KUKA KRL program: MyProgram_124().src

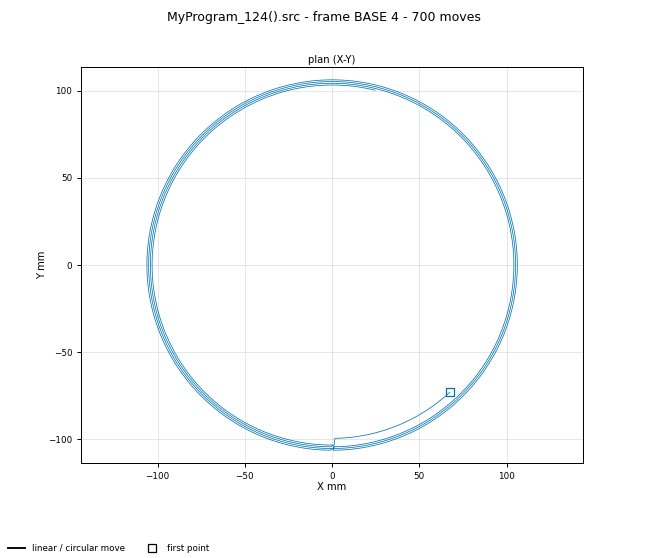
[picture p0: tool path of MyProgram_124().src in frame BASE 4, 700 of 700 moves have a stored position in this frame; points joined in program order, loops and branches not executed]
&ACCESS RVP
&REL 1
&PARAM TEMPLATE = C:\KRC\Roboter\Template\vorgabe
&PARAM EDITMASK = *
DEF MyProgram_124()
; ---- Setting reference (Base) ----
$BASE = BASE_DATA[4]

; --------------------------
; ---- Setting tool (TCP) ----
$TOOL = TOOL_DATA[3]
; --------------------------

$VEL.CP = VEL_APROX_PRINT
Startdeposition()
$VEL.CP = VEL_PRINT
LIN {X 67.4636,Y -72.9151,Z 103,A -51.9961,B 24.9391,C -1.8028,E1 25.1077,E2 497.4549} C_DIS
LIN {X 64.8778,Y -75.2264,Z 103,A -54.0592,B 24.9396,C -1.7957,E1 25.1034,E2 499.5265} C_DIS
LIN {X 62.0723,Y -77.5576,Z 103,A -56.1658,B 24.9399,C -1.791,E1 25.0988,E2 501.6364} C_DIS
LIN {X 59.4843,Y -79.5578,Z 103,A -57.817,B 24.9395,C -1.7961,E1 25.0952,E2 503.2694} C_DIS
LIN {X 57.5377,Y -80.9767,Z 103,A -59.2001,B 24.9397,C -1.7935,E1 25.092,E2 504.6539} C_DIS
LIN {X 55.1858,Y -82.5995,Z 103,A -61.0068,B 24.9403,C -1.784,E1 25.0878,E2 506.4769} C_DIS
LIN {X 52.4682,Y -84.3499,Z 103,A -62.7627,B 24.9403,C -1.7846,E1 25.0837,E2 508.2256} C_DIS
LIN {X 50.0146,Y -85.8293,Z 103,A -64.3819,B 24.9404,C -1.7828,E1 25.0798,E2 509.8441} C_DIS
LIN {X 47.8461,Y -87.0565,Z 103,A -65.9289,B 24.9409,C -1.7761,E1 25.076,E2 511.4025} C_DIS
LIN {X 45.0141,Y -88.5525,Z 103,A -67.6742,B 24.9409,C -1.7769,E1 25.0717,E2 513.141} C_DIS
LIN {X 42.0972,Y -89.9758,Z 103,A -69.5826,B 24.9411,C -1.7725,E1 25.0669,E2 515.0548} C_DIS
LIN {X 39.1268,Y -91.3084,Z 103,A -71.5179,B 24.9415,C -1.7674,E1 25.0619,E2 516.9974} C_DIS
LIN {X 36.1356,Y -92.5313,Z 103,A -73.2136,B 24.9412,C -1.7713,E1 25.0575,E2 518.6802} C_DIS
LIN {X 33.7277,Y -93.4362,Z 103,A -74.6858,B 24.9413,C -1.7697,E1 25.0537,E2 520.153} C_DIS
LIN {X 31.1034,Y -94.3433,Z 103,A -76.4427,B 24.9418,C -1.7618,E1 25.049,E2 521.9253} C_DIS
LIN {X 28.0406,Y -95.2971,Z 103,A -78.1345,B 24.9416,C -1.7657,E1 25.0445,E2 523.6049} C_DIS
LIN {X 25.3105,Y -96.06,Z 103,A -79.7633,B 24.9416,C -1.7641,E1 25.0401,E2 525.2347} C_DIS
LIN {X 22.5573,Y -96.7418,Z 103,A -81.5,B 24.942,C -1.7587,E1 25.0354,E2 526.9817} C_DIS
LIN {X 19.9429,Y -97.3142,Z 103,A -83.0396,B 24.9421,C -1.7575,E1 25.0312,E2 528.5221} C_DIS
LIN {X 16.9823,Y -97.8762,Z 103,A -84.8399,B 24.9424,C -1.7538,E1 25.0262,E2 530.3294} C_DIS
LIN {X 13.8632,Y -98.3646,Z 103,A -86.5531,B 24.9422,C -1.7565,E1 25.0215,E2 532.0345} C_DIS
LIN {X 10.9392,Y -98.7343,Z 103,A -88.1902,B 24.9421,C -1.7578,E1 25.017,E2 533.6673} C_DIS
LIN {X 8.1007,Y -99.006,Z 103,A -89.9343,B 24.9424,C -1.7533,E1 25.0121,E2 535.4211} C_DIS
LIN {X 4.8754,Y -99.2188,Z 103,A -91.8612,B 24.9426,C -1.7502,E1 25.0067,E2 537.3547} C_DIS
LIN {X 1.6447,Y -99.3232,Z 103,A -93.5925,B 24.9423,C -1.7545,E1 25.0019,E2 539.0753} C_DIS
LIN {X 1.6447,Y -99.3232,Z 103,A -93.5925,B 24.9423,C -1.7545,E1 25.0019,E2 539.0753} C_DIS
Enddeposition()
LIN {X 0.7394,Y -106.1621,Z 104,A -93.403,B 24.9477,C -1.6702,E1 25.0019,E2 539.0857} C_DIS
Startdeposition()
$VEL.CP = VEL_PRINT
LIN {X 4.4145,Y -106.0742,Z 104,A -91.2125,B 24.9472,C -1.6792,E1 25.008,E2 536.8744} C_DIS
LIN {X 7.8102,Y -105.8803,Z 104,A -89.2631,B 24.9468,C -1.6846,E1 25.0135,E2 534.913} C_DIS
LIN {X 10.7746,Y -105.6181,Z 104,A -87.8003,B 24.9471,C -1.6797,E1 25.0175,E2 533.4628} C_DIS
LIN {X 14.6548,Y -105.15,Z 104,A -85.7013,B 24.9471,C -1.6806,E1 25.0233,E2 531.3633} C_DIS
LIN {X 18.1507,Y -104.6049,Z 104,A -83.6459,B 24.9466,C -1.688,E1 25.0291,E2 529.2925} C_DIS
LIN {X 20.7123,Y -104.128,Z 104,A -82.2422,B 24.9466,C -1.6891,E1 25.0329,E2 527.8878} C_DIS
LIN {X 23.5206,Y -103.5284,Z 104,A -80.7997,B 24.9467,C -1.6861,E1 25.0368,E2 526.4542} C_DIS
LIN {X 25.7967,Y -102.9862,Z 104,A -79.5774,B 24.9467,C -1.6857,E1 25.0401,E2 525.2348} C_DIS
LIN {X 28.3163,Y -102.3221,Z 104,A -78.0325,B 24.9463,C -1.6929,E1 25.0443,E2 523.6752} C_DIS
LIN {X 30.8189,Y -101.5964,Z 104,A -76.7716,B 24.9466,C -1.6885,E1 25.0477,E2 522.427} C_DIS
LIN {X 33.6539,Y -100.6911,Z 104,A -75.0798,B 24.9462,C -1.6941,E1 25.0522,E2 520.7253} C_DIS
LIN {X 36.9909,Y -99.5153,Z 104,A -73.1238,B 24.9459,C -1.6985,E1 25.0573,E2 518.7628} C_DIS
LIN {X 40.6287,Y -98.0864,Z 104,A -71.1625,B 24.9461,C -1.6953,E1 25.0624,E2 516.8135} C_DIS
LIN {X 43.0236,Y -97.0598,Z 104,A -69.761,B 24.9461,C -1.6972,E1 25.066,E2 515.4108} C_DIS
LIN {X 45.3926,Y -95.9747,Z 104,A -68.3595,B 24.9459,C -1.6993,E1 25.0695,E2 514.0081} C_DIS
LIN {X 48.0641,Y -94.6632,Z 104,A -66.7592,B 24.9457,C -1.7017,E1 25.0735,E2 512.4063} C_DIS
LIN {X 51.1925,Y -93.0106,Z 104,A -64.7153,B 24.9452,C -1.7106,E1 25.0786,E2 510.3472} C_DIS
LIN {X 53.7785,Y -91.5378,Z 104,A -63.2568,B 24.9454,C -1.7074,E1 25.0821,E2 508.9008} C_DIS
LIN {X 56.0305,Y -90.1768,Z 104,A -61.8515,B 24.9452,C -1.7094,E1 25.0854,E2 507.4951} C_DIS
LIN {X 59.2904,Y -88.0678,Z 104,A -59.7558,B 24.945,C -1.7136,E1 25.0903,E2 505.3965} C_DIS
LIN {X 61.4338,Y -86.5862,Z 104,A -58.356,B 24.9448,C -1.7162,E1 25.0935,E2 503.9954} C_DIS
LIN {X 63.5403,Y -85.0524,Z 104,A -56.9295,B 24.9446,C -1.72,E1 25.0967,E2 502.565} C_DIS
LIN {X 65.6084,Y -83.4675,Z 104,A -55.5565,B 24.9445,C -1.7216,E1 25.0998,E2 501.1931} C_DIS
LIN {X 67.6371,Y -81.8322,Z 104,A -54.1568,B 24.9443,C -1.7245,E1 25.1028,E2 499.792} C_DIS
LIN {X 69.625,Y -80.1477,Z 104,A -52.7579,B 24.9441,C -1.7274,E1 25.1058,E2 498.3917} C_DIS
LIN {X 71.5709,Y -78.4149,Z 104,A -51.3584,B 24.9439,C -1.7304,E1 25.1087,E2 496.9908} C_DIS
LIN {X 74.4086,Y -75.7274,Z 104,A -49.4414,B 24.9441,C -1.7272,E1 25.1125,E2 495.0891} C_DIS
LIN {X 76.2447,Y -73.8785,Z 104,A -48.0425,B 24.9439,C -1.7304,E1 25.1153,E2 493.6888} C_DIS
LIN {X 77.7844,Y -72.258,Z 104,A -46.6614,B 24.9432,C -1.7409,E1 25.1179,E2 492.2889} C_DIS
LIN {X 79.5343,Y -70.3273,Z 104,A -45.2623,B 24.943,C -1.7441,E1 25.1205,E2 490.8884} C_DIS
LIN {X 81.5346,Y -67.9952,Z 104,A -43.8429,B 24.9434,C -1.7383,E1 25.1231,E2 489.4892} C_DIS
LIN {X 82.8893,Y -66.34,Z 104,A -42.4537,B 24.9425,C -1.7514,E1 25.1256,E2 488.0756} C_DIS
LIN {X 84.4924,Y -64.2859,Z 104,A -41.068,B 24.9423,C -1.7543,E1 25.1279,E2 486.6896} C_DIS
LIN {X 86.0446,Y -62.193,Z 104,A -39.6701,B 24.9421,C -1.7578,E1 25.1302,E2 485.2901} C_DIS
LIN {X 87.79,Y -59.7006,Z 104,A -38.061,B 24.9419,C -1.761,E1 25.1328,E2 483.6814} C_DIS
LIN {X 89.8926,Y -56.4855,Z 104,A -36.1587,B 24.9419,C -1.7595,E1 25.1356,E2 481.7921} C_DIS
LIN {X 91.0633,Y -54.5812,Z 104,A -34.7784,B 24.9413,C -1.7705,E1 25.1377,E2 480.3931} C_DIS
LIN {X 92.5559,Y -52.0066,Z 104,A -33.1821,B 24.941,C -1.7747,E1 25.1399,E2 478.7949} C_DIS
LIN {X 94.2389,Y -48.8944,Z 104,A -31.1438,B 24.9402,C -1.786,E1 25.1426,E2 476.7409} C_DIS
LIN {X 95.5708,Y -46.2332,Z 104,A -29.6891,B 24.9403,C -1.7842,E1 25.1444,E2 475.298} C_DIS
LIN {X 96.6964,Y -43.83,Z 104,A -28.283,B 24.9401,C -1.7875,E1 25.146,E2 473.8919} C_DIS
LIN {X 97.7242,Y -41.488,Z 104,A -26.8064,B 24.9396,C -1.7959,E1 25.1476,E2 472.4035} C_DIS
LIN {X 98.9185,Y -38.554,Z 104,A -25.1568,B 24.9394,C -1.7985,E1 25.1493,E2 470.7568} C_DIS
LIN {X 99.9618,Y -35.7669,Z 104,A -23.6014,B 24.9392,C -1.8013,E1 25.1508,E2 469.2036} C_DIS
LIN {X 100.9235,Y -32.9506,Z 104,A -22.0063,B 24.9389,C -1.8059,E1 25.1522,E2 467.6066} C_DIS
LIN {X 102.0679,Y -29.2135,Z 104,A -19.9111,B 24.9385,C -1.812,E1 25.1539,E2 465.5091} C_DIS
LIN {X 102.9862,Y -25.7967,Z 104,A -17.8737,B 24.9377,C -1.8236,E1 25.1554,E2 463.4561} C_DIS
LIN {X 103.5883,Y -23.2615,Z 104,A -16.4771,B 24.9374,C -1.8277,E1 25.1562,E2 462.0579} C_DIS
LIN {X 104.1964,Y -20.3566,Z 104,A -15.0246,B 24.9374,C -1.8263,E1 25.157,E2 460.617} C_DIS
LIN {X 104.666,Y -17.7854,Z 104,A -13.6266,B 24.9372,C -1.8303,E1 25.1577,E2 459.2178} C_DIS
LIN {X 105.2497,Y -13.9209,Z 104,A -11.7135,B 24.9373,C -1.8287,E1 25.1585,E2 457.3199} C_DIS
LIN {X 105.5491,Y -11.4338,Z 104,A -10.118,B 24.9363,C -1.8436,E1 25.159,E2 455.6986} C_DIS
LIN {X 105.8803,Y -7.8102,Z 104,A -8.0982,B 24.9357,C -1.8524,E1 25.1595,E2 453.6701} C_DIS
LIN {X 106.0401,Y -5.2094,Z 104,A -6.7017,B 24.9354,C -1.8565,E1 25.1597,E2 452.2721} C_DIS
LIN {X 106.1531,Y -1.6731,Z 104,A -4.7932,B 24.935,C -1.8627,E1 25.1597,E2 450.3604} C_DIS
LIN {X 106.136,Y 2.6055,Z 104,A -2.5124,B 24.9345,C -1.8689,E1 25.1597,E2 448.0787} C_DIS
LIN {X 106.0401,Y 5.2094,Z 104,A -1.1158,B 24.9342,C -1.873,E1 25.1595,E2 446.6806} C_DIS
LIN {X 105.8803,Y 7.8102,Z 104,A 0.2806,B 24.934,C -1.8771,E1 25.1592,E2 445.2829} C_DIS
LIN {X 105.5211,Y 11.7021,Z 104,A 2.4327,B 24.9333,C -1.8857,E1 25.1586,E2 443.1232} C_DIS
LIN {X 105.0188,Y 15.5781,Z 104,A 4.3294,B 24.9335,C -1.8831,E1 25.1579,E2 441.2437} C_DIS
LIN {X 104.6049,Y 18.1507,Z 104,A 5.8673,B 24.9328,C -1.8933,E1 25.1572,E2 439.6909} C_DIS
LIN {X 104.0535,Y 21.0751,Z 104,A 7.3213,B 24.9329,C -1.8917,E1 25.1564,E2 438.249} C_DIS
LIN {X 103.2072,Y 24.8908,Z 104,A 9.2641,B 24.9329,C -1.8911,E1 25.1552,E2 436.3189} C_DIS
LIN {X 102.6619,Y 27.0586,Z 104,A 10.7562,B 24.9318,C -1.9071,E1 25.1542,E2 434.7977} C_DIS
LIN {X 101.8958,Y 29.8097,Z 104,A 12.0237,B 24.9323,C -1.9,E1 25.1532,E2 433.5542} C_DIS
LIN {X 101.2105,Y 32.0633,Z 104,A 13.4091,B 24.9317,C -1.9088,E1 25.152,E2 432.156} C_DIS
LIN {X 100.3932,Y 34.5375,Z 104,A 14.9476,B 24.931,C -1.9187,E1 25.1506,E2 430.6028} C_DIS
LIN {X 99.3842,Y 37.3372,Z 104,A 16.4024,B 24.9311,C -1.917,E1 25.1493,E2 429.1602} C_DIS
LIN {X 98.5433,Y 39.5062,Z 104,A 17.6053,B 24.9311,C -1.9184,E1 25.148,E2 427.9607} C_DIS
LIN {X 97.5296,Y 41.9459,Z 104,A 19.0045,B 24.9308,C -1.9214,E1 25.1465,E2 426.562} C_DIS
LIN {X 96.5245,Y 44.2115,Z 104,A 20.5441,B 24.9299,C -1.9338,E1 25.1447,E2 425.0014} C_DIS
LIN {X 95.4104,Y 46.567,Z 104,A 21.7939,B 24.9301,C -1.9311,E1 25.1432,E2 423.7647} C_DIS
LIN {X 94.2389,Y 48.8944,Z 104,A 23.1917,B 24.9298,C -1.9347,E1 25.1414,E2 422.366} C_DIS
LIN {X 92.83,Y 51.5158,Z 104,A 24.7883,B 24.9295,C -1.9387,E1 25.1393,E2 420.7683} C_DIS
LIN {X 90.8019,Y 55.0114,Z 104,A 26.9328,B 24.9292,C -1.943,E1 25.1363,E2 418.6247} C_DIS
LIN {X 88.9926,Y 57.896,Z 104,A 28.7841,B 24.9288,C -1.9483,E1 25.1335,E2 416.7701} C_DIS
LIN {X 87.3336,Y 60.3667,Z 104,A 30.3816,B 24.9286,C -1.9521,E1 25.131,E2 415.1715} C_DIS
LIN {X 85.2749,Y 63.2442,Z 104,A 32.2808,B 24.9282,C -1.9564,E1 25.1278,E2 413.2714} C_DIS
LIN {X 83.6971,Y 65.3179,Z 104,A 33.6798,B 24.928,C -1.9595,E1 25.1255,E2 411.8716} C_DIS
LIN {X 81.8322,Y 67.6371,Z 104,A 35.2776,B 24.9278,C -1.963,E1 25.1226,E2 410.273} C_DIS
LIN {X 80.2103,Y 69.5532,Z 104,A 36.6598,B 24.9274,C -1.9673,E1 25.1201,E2 408.8869} C_DIS
LIN {X 78.6653,Y 71.298,Z 104,A 37.8771,B 24.9274,C -1.9684,E1 25.1179,E2 407.6724} C_DIS
LIN {X 76.8918,Y 73.2071,Z 104,A 39.2766,B 24.9271,C -1.9713,E1 25.1152,E2 406.2723} C_DIS
LIN {X 74.8086,Y 75.3323,Z 104,A 40.6937,B 24.9275,C -1.9668,E1 25.1124,E2 404.8717} C_DIS
LIN {X 73.2071,Y 76.8918,Z 104,A 42.0765,B 24.9267,C -1.9767,E1 25.1096,E2 403.4713} C_DIS
LIN {X 71.0221,Y 78.9123,Z 104,A 43.6753,B 24.9265,C -1.9797,E1 25.1063,E2 401.8719} C_DIS
LIN {X 68.0694,Y 81.4729,Z 104,A 45.8349,B 24.9261,C -1.9859,E1 25.1017,E2 399.706} C_DIS
LIN {X 65.3179,Y 83.6971,Z 104,A 47.8193,B 24.9256,C -1.9925,E1 25.0974,E2 397.7134} C_DIS
LIN {X 63.2442,Y 85.2749,Z 104,A 49.0899,B 24.9258,C -1.9894,E1 25.0945,E2 396.4548} C_DIS
LIN {X 61.1324,Y 86.8013,Z 104,A 50.4796,B 24.9257,C -1.9911,E1 25.0914,E2 395.0658} C_DIS
LIN {X 58.6746,Y 88.4793,Z 104,A 52.08,B 24.9255,C -1.9935,E1 25.0877,E2 393.4651} C_DIS
LIN {X 56.4855,Y 89.8926,Z 104,A 53.5325,B 24.9252,C -1.9976,E1 25.0842,E2 392.0076} C_DIS
LIN {X 53.4596,Y 91.7262,Z 104,A 55.5266,B 24.9247,C -2.0039,E1 25.0794,E2 390.0048} C_DIS
LIN {X 50.0472,Y 93.6318,Z 104,A 57.6296,B 24.9245,C -2.0066,E1 25.0743,E2 387.9015} C_DIS
LIN {X 47.7343,Y 94.8318,Z 104,A 58.8901,B 24.9248,C -2.0024,E1 25.0712,E2 386.6544} C_DIS
LIN {X 45.3926,Y 95.9747,Z 104,A 60.4347,B 24.9243,C -2.0098,E1 25.0673,E2 385.0964} C_DIS
LIN {X 42.6841,Y 97.2078,Z 104,A 61.8947,B 24.9246,C -2.0057,E1 25.0636,E2 383.6497} C_DIS
LIN {X 39.9794,Y 98.3507,Z 104,A 63.5207,B 24.9243,C -2.009,E1 25.0594,E2 382.0195} C_DIS
LIN {X 36.9909,Y 99.5153,Z 104,A 65.3455,B 24.9239,C -2.0145,E1 25.0546,E2 380.1857} C_DIS
LIN {X 34.1866,Y 100.5115,Z 104,A 66.8064,B 24.9242,C -2.01,E1 25.0508,E2 378.7384} C_DIS
LIN {X 31.6232,Y 101.347,Z 104,A 68.32,B 24.924,C -2.0135,E1 25.0467,E2 377.2192} C_DIS
LIN {X 28.6727,Y 102.2212,Z 104,A 70.0997,B 24.9235,C -2.0195,E1 25.0419,E2 375.4283} C_DIS
LIN {X 25.7967,Y 102.9862,Z 104,A 71.6633,B 24.9235,C -2.0187,E1 25.0377,E2 373.8689} C_DIS
LIN {X 23.2615,Y 103.5883,Z 104,A 72.9259,B 24.924,C -2.0137,E1 25.0343,E2 372.62} C_DIS
LIN {X 20.7123,Y 104.128,Z 104,A 74.473,B 24.9235,C -2.02,E1 25.03,E2 371.06} C_DIS
LIN {X 17.7854,Y 104.666,Z 104,A 75.9356,B 24.9239,C -2.0149,E1 25.026,E2 369.611} C_DIS
LIN {X 15.0661,Y 105.0916,Z 104,A 77.3709,B 24.9239,C -2.0133,E1 25.0221,E2 368.1808} C_DIS
LIN {X 12.6898,Y 105.4054,Z 104,A 78.561,B 24.9243,C -2.0094,E1 25.0188,E2 367.0007} C_DIS
LIN {X 10.4063,Y 105.6567,Z 104,A 80.0948,B 24.9234,C -2.0213,E1 25.0145,E2 365.44} C_DIS
LIN {X 7.8102,Y 105.8803,Z 104,A 81.5009,B 24.9234,C -2.0213,E1 25.0106,E2 364.0343} C_DIS
LIN {X 5.2094,Y 106.0401,Z 104,A 82.9074,B 24.9234,C -2.0213,E1 25.0066,E2 362.6285} C_DIS
LIN {X 1.8879,Y 106.1492,Z 104,A 84.6484,B 24.9236,C -2.0191,E1 25.0018,E2 360.8931} C_DIS
LIN {X -1.6731,Y 106.1531,Z 104,A 86.4353,B 24.924,C -2.0133,E1 24.9968,E2 359.1198} C_DIS
LIN {X -4.2778,Y 106.0801,Z 104,A 87.7061,B 24.9244,C -2.0076,E1 24.9933,E2 357.8624} C_DIS
LIN {X -6.8798,Y 105.9432,Z 104,A 89.2303,B 24.9241,C -2.0117,E1 24.9891,E2 356.328} C_DIS
LIN {X -9.4777,Y 105.7424,Z 104,A 90.704,B 24.924,C -2.0137,E1 24.9849,E2 354.8489} C_DIS
LIN {X -12.9961,Y 105.3695,Z 104,A 92.7585,B 24.9236,C -2.0182,E1 24.9792,E2 352.7824} C_DIS
LIN {X -15.5781,Y 105.0188,Z 104,A 94.0241,B 24.9241,C -2.0118,E1 24.9758,E2 351.5309} C_DIS
LIN {X -18.5419,Y 104.5345,Z 104,A 95.6379,B 24.9242,C -2.0104,E1 24.9713,E2 349.9189} C_DIS
LIN {X -22.3504,Y 103.787,Z 104,A 97.563,B 24.9248,C -2.0021,E1 24.9661,E2 348.0113} C_DIS
LIN {X -24.531,Y 103.295,Z 104,A 98.9549,B 24.9244,C -2.0081,E1 24.9623,E2 346.6032} C_DIS
LIN {X -27.0586,Y 102.6619,Z 104,A 100.364,B 24.9244,C -2.0068,E1 24.9585,E2 345.1952} C_DIS
LIN {X -29.9249,Y 101.8616,Z 104,A 101.7911,B 24.9251,C -1.9983,E1 24.9547,E2 343.7862} C_DIS
LIN {X -32.0633,Y 101.2105,Z 104,A 103.3676,B 24.9242,C -2.0111,E1 24.9504,E2 342.1765} C_DIS
LIN {X -34.887,Y 100.2706,Z 104,A 104.7938,B 24.9248,C -2.0022,E1 24.9467,E2 340.7686} C_DIS
LIN {X -38.554,Y 98.9185,Z 104,A 106.726,B 24.9255,C -1.9927,E1 24.9417,E2 338.8551} C_DIS
LIN {X -40.7938,Y 98.0168,Z 104,A 108.2418,B 24.9251,C -1.9989,E1 24.9377,E2 337.321} C_DIS
LIN {X -43.0236,Y 97.0598,Z 104,A 109.6727,B 24.9249,C -2.0016,E1 24.934,E2 335.8803} C_DIS
LIN {X -45.3926,Y 95.9747,Z 104,A 110.9409,B 24.9254,C -1.9942,E1 24.9308,E2 334.6266} C_DIS
LIN {X -48.0641,Y 94.6632,Z 104,A 112.5526,B 24.9256,C -1.9918,E1 24.9268,E2 333.0162} C_DIS
LIN {X -51.1925,Y 93.0106,Z 104,A 114.6121,B 24.9254,C -1.9942,E1 24.9217,E2 330.9453} C_DIS
LIN {X -54.5812,Y 91.0633,Z 104,A 116.5866,B 24.9261,C -1.9854,E1 24.917,E2 328.9859} C_DIS
LIN {X -57.1113,Y 89.4963,Z 104,A 118.0161,B 24.9268,C -1.9757,E1 24.9137,E2 327.5748} C_DIS
LIN {X -59.2904,Y 88.0678,Z 104,A 119.612,B 24.9265,C -1.9801,E1 24.9099,E2 325.9632} C_DIS
LIN {X -61.4338,Y 86.5862,Z 104,A 121.0241,B 24.9267,C -1.9775,E1 24.9067,E2 324.5525} C_DIS
LIN {X -64.5792,Y 84.2663,Z 104,A 123.1434,B 24.927,C -1.9735,E1 24.9019,E2 322.4353} C_DIS
LIN {X -67.3522,Y 82.0689,Z 104,A 125.2047,B 24.9269,C -1.9749,E1 24.8974,E2 320.3627} C_DIS
LIN {X -69.346,Y 80.3913,Z 104,A 126.6177,B 24.9271,C -1.972,E1 24.8944,E2 318.9512} C_DIS
LIN {X -71.5709,Y 78.4149,Z 104,A 128.0891,B 24.9277,C -1.9633,E1 24.8914,E2 317.4946} C_DIS
LIN {X -74.1452,Y 75.9877,Z 104,A 130.1963,B 24.9275,C -1.9661,E1 24.8871,E2 315.372} C_DIS
LIN {X -76.2447,Y 73.8785,Z 104,A 131.6232,B 24.9283,C -1.9556,E1 24.8844,E2 313.9641} C_DIS
LIN {X -78.6653,Y 71.298,Z 104,A 133.6864,B 24.9283,C -1.9565,E1 24.8805,E2 311.8898} C_DIS
LIN {X -80.3913,Y 69.346,Z 104,A 134.9937,B 24.9288,C -1.9492,E1 24.8781,E2 310.5939} C_DIS
LIN {X -82.0689,Y 67.3522,Z 104,A 136.3717,B 24.9291,C -1.9445,E1 24.8756,E2 309.2208} C_DIS
LIN {X -83.9232,Y 65.0245,Z 104,A 137.803,B 24.9299,C -1.9338,E1 24.8732,E2 307.8081} C_DIS
LIN {X -85.2749,Y 63.2442,Z 104,A 139.2004,B 24.9296,C -1.9375,E1 24.8708,E2 306.3951} C_DIS
LIN {X -86.8013,Y 61.1324,Z 104,A 140.7581,B 24.9295,C -1.9392,E1 24.8683,E2 304.8257} C_DIS
LIN {X -88.9926,Y 57.896,Z 104,A 142.8804,B 24.9299,C -1.9338,E1 24.865,E2 302.7058} C_DIS
LIN {X -90.579,Y 55.3781,Z 104,A 144.3533,B 24.9306,C -1.9244,E1 24.8629,E2 301.2478} C_DIS
LIN {X -92.3753,Y 52.33,Z 104,A 146.2751,B 24.9309,C -1.9193,E1 24.8602,E2 299.3282} C_DIS
LIN {X -93.8043,Y 49.7195,Z 104,A 147.7073,B 24.9317,C -1.9083,E1 24.8583,E2 297.9147} C_DIS
LIN {X -94.8318,Y 47.7343,Z 104,A 149.1055,B 24.9315,C -1.9117,E1 24.8565,E2 296.5009} C_DIS
LIN {X -96.131,Y 45.0569,Z 104,A 150.5383,B 24.9323,C -1.9006,E1 24.8548,E2 295.0868} C_DIS
LIN {X -97.0598,Y 43.0236,Z 104,A 152.1061,B 24.9316,C -1.91,E1 24.853,E2 293.4878} C_DIS
LIN {X -98.5776,Y 39.422,Z 104,A 154.06,B 24.9325,C -1.8979,E1 24.8509,E2 291.5519} C_DIS
LIN {X -99.5154,Y 36.9909,Z 104,A 155.6192,B 24.9324,C -1.8992,E1 24.8494,E2 289.981} C_DIS
LIN {X -100.8094,Y 33.3029,Z 104,A 157.5996,B 24.9332,C -1.8879,E1 24.8476,E2 288.0163} C_DIS
LIN {X -101.7485,Y 30.306,Z 104,A 159.2508,B 24.9337,C -1.881,E1 24.8462,E2 286.3719} C_DIS
LIN {X -102.4187,Y 27.9588,Z 104,A 160.6325,B 24.9338,C -1.8792,E1 24.8452,E2 284.9866} C_DIS
LIN {X -103.3784,Y 24.1701,Z 104,A 162.5727,B 24.9347,C -1.8663,E1 24.8439,E2 283.0658} C_DIS
LIN {X -103.8659,Y 21.9886,Z 104,A 164.0947,B 24.9342,C -1.8739,E1 24.843,E2 281.5167} C_DIS
LIN {X -104.4398,Y 19.0685,Z 104,A 165.5887,B 24.9348,C -1.8647,E1 24.8422,E2 280.0357} C_DIS
LIN {X -105.0188,Y 15.5781,Z 104,A 167.5117,B 24.9352,C -1.859,E1 24.8414,E2 278.1149} C_DIS
LIN {X -105.4126,Y 12.6282,Z 104,A 168.9452,B 24.936,C -1.8476,E1 24.8409,E2 276.7001} C_DIS
LIN {X -105.6567,Y 10.4063,Z 104,A 170.4872,B 24.9354,C -1.8558,E1 24.8404,E2 275.1291} C_DIS
LIN {X -105.8803,Y 7.8102,Z 104,A 171.9034,B 24.9357,C -1.8517,E1 24.8401,E2 273.7143} C_DIS
LIN {X -106.0401,Y 5.2094,Z 104,A 173.3197,B 24.936,C -1.8475,E1 24.8399,E2 272.2995} C_DIS
LIN {X -106.136,Y 2.6055,Z 104,A 174.5924,B 24.9367,C -1.8381,E1 24.8399,E2 271.0416} C_DIS
LIN {X -106.1663,Y -0.3058,Z 104,A 176.2085,B 24.9369,C -1.8346,E1 24.8398,E2 269.4239} C_DIS
LIN {X -106.0801,Y -4.2778,Z 104,A 178.1502,B 24.9379,C -1.8204,E1 24.8399,E2 267.5045} C_DIS
LIN {X -105.9432,Y -6.8798,Z 104,A 179.5665,B 24.9382,C -1.8162,E1 24.8402,E2 266.0896} C_DIS
LIN {X -105.7424,Y -9.4777,Z 104,A -178.8337,B 24.938,C -1.8188,E1 24.8405,E2 264.4741} C_DIS
LIN {X -105.478,Y -12.0699,Z 104,A -177.361,B 24.9381,C -1.8167,E1 24.841,E2 262.9975} C_DIS
LIN {X -105.0188,Y -15.5781,Z 104,A -175.4949,B 24.9387,C -1.8091,E1 24.8417,E2 261.1386} C_DIS
LIN {X -104.6049,Y -18.1507,Z 104,A -173.9358,B 24.9386,C -1.8102,E1 24.8424,E2 259.5674} C_DIS
LIN {X -104.128,Y -20.7123,Z 104,A -172.5134,B 24.9388,C -1.8064,E1 24.8432,E2 258.1458} C_DIS
LIN {X -103.5883,Y -23.2615,Z 104,A -171.1041,B 24.9391,C -1.8022,E1 24.844,E2 256.7383} C_DIS
LIN {X -102.9862,Y -25.7967,Z 104,A -169.8317,B 24.9397,C -1.7929,E1 24.8449,E2 255.4804} C_DIS
LIN {X -102.3221,Y -28.3163,Z 104,A -168.2727,B 24.9397,C -1.7942,E1 24.846,E2 253.9093} C_DIS
LIN {X -101.5964,Y -30.8189,Z 104,A -167.0005,B 24.9403,C -1.785,E1 24.847,E2 252.6517} C_DIS
LIN {X -100.6911,Y -33.6539,Z 104,A -165.3839,B 24.9406,C -1.7806,E1 24.8484,E2 251.0363} C_DIS
LIN {X -99.5153,Y -36.9909,Z 104,A -163.3114,B 24.9406,C -1.781,E1 24.8504,E2 248.9513} C_DIS
LIN {X -98.0864,Y -40.6287,Z 104,A -161.339,B 24.9413,C -1.7698,E1 24.8524,E2 246.9946} C_DIS
LIN {X -97.0598,Y -43.0236,Z 104,A -159.9039,B 24.9415,C -1.7668,E1 24.854,E2 245.5587} C_DIS
LIN {X -95.9747,Y -45.3926,Z 104,A -158.5092,B 24.9418,C -1.7624,E1 24.8557,E2 244.1669} C_DIS
LIN {X -94.6632,Y -48.0641,Z 104,A -156.8933,B 24.9421,C -1.7583,E1 24.8577,E2 242.5521} C_DIS
LIN {X -93.0106,Y -51.1925,Z 104,A -154.8294,B 24.9421,C -1.7588,E1 24.8604,E2 240.4761} C_DIS
LIN {X -91.5378,Y -53.7785,Z 104,A -153.3321,B 24.9426,C -1.7504,E1 24.8625,E2 238.9908} C_DIS
LIN {X -89.4963,Y -57.1113,Z 104,A -151.419,B 24.9434,C -1.7376,E1 24.8653,E2 237.0986} C_DIS
LIN {X -88.0678,Y -59.2904,Z 104,A -149.8211,B 24.9432,C -1.7411,E1 24.8678,E2 235.4843} C_DIS
LIN {X -86.5862,Y -61.4338,Z 104,A -148.4075,B 24.9434,C -1.7379,E1 24.8701,E2 234.0714} C_DIS
LIN {X -84.8783,Y -63.7721,Z 104,A -146.9035,B 24.9438,C -1.7318,E1 24.8725,E2 232.5746} C_DIS
LIN {X -83.4675,Y -65.6084,Z 104,A -145.58,B 24.9438,C -1.7316,E1 24.8748,E2 231.2455} C_DIS
LIN {X -81.8322,Y -67.6371,Z 104,A -144.1664,B 24.944,C -1.7285,E1 24.8773,E2 229.8325} C_DIS
LIN {X -80.1477,Y -69.625,Z 104,A -142.7535,B 24.9442,C -1.7255,E1 24.8799,E2 228.4203} C_DIS
LIN {X -78.4149,Y -71.5709,Z 104,A -141.34,B 24.9444,C -1.7226,E1 24.8825,E2 227.0075} C_DIS
LIN {X -76.5611,Y -73.5502,Z 104,A -139.9058,B 24.9447,C -1.7183,E1 24.8853,E2 225.5773} C_DIS
LIN {X -73.8785,Y -76.2447,Z 104,A -137.9913,B 24.9453,C -1.7088,E1 24.889,E2 223.6774} C_DIS
LIN {X -72.258,Y -77.7844,Z 104,A -136.5963,B 24.945,C -1.7134,E1 24.8919,E2 222.2657} C_DIS
LIN {X -70.3273,Y -79.5343,Z 104,A -135.1835,B 24.9451,C -1.7109,E1 24.8949,E2 220.8532} C_DIS
LIN {X -68.2918,Y -81.2881,Z 104,A -133.7062,B 24.9453,C -1.7091,E1 24.898,E2 219.3744} C_DIS
LIN {X -66.34,Y -82.8893,Z 104,A -132.3599,B 24.9455,C -1.706,E1 24.9009,E2 218.0304} C_DIS
LIN {X -64.2859,Y -84.4924,Z 104,A -130.948,B 24.9456,C -1.7037,E1 24.904,E2 216.6189} C_DIS
LIN {X -62.193,Y -86.0446,Z 104,A -129.5365,B 24.9457,C -1.7015,E1 24.9072,E2 215.2078} C_DIS
LIN {X -60.0626,Y -87.5449,Z 104,A -127.9381,B 24.9454,C -1.7065,E1 24.9109,E2 213.5919} C_DIS
LIN {X -57.7425,Y -89.0912,Z 104,A -126.5456,B 24.9459,C -1.6999,E1 24.9142,E2 212.2107} C_DIS
LIN {X -55.6946,Y -90.3866,Z 104,A -125.303,B 24.9461,C -1.6953,E1 24.9171,E2 210.9749} C_DIS
LIN {X -53.4596,Y -91.7262,Z 104,A -123.7501,B 24.9459,C -1.699,E1 24.9209,E2 209.4087} C_DIS
LIN {X -50.0472,Y -93.6318,Z 104,A -121.6357,B 24.9461,C -1.6963,E1 24.926,E2 207.2946} C_DIS
LIN {X -47.4025,Y -94.9963,Z 104,A -120.1665,B 24.9465,C -1.689,E1 24.9297,E2 205.8388} C_DIS
LIN {X -45.0569,Y -96.131,Z 104,A -118.7015,B 24.9465,C -1.6897,E1 24.9334,E2 204.3686} C_DIS
LIN {X -42.6841,Y -97.2078,Z 104,A -117.3472,B 24.9467,C -1.6861,E1 24.9368,E2 203.0195} C_DIS
LIN {X -39.422,Y -98.5776,Z 104,A -115.2907,B 24.9465,C -1.6899,E1 24.9422,E2 200.9494} C_DIS
LIN {X -36.9909,Y -99.5153,Z 104,A -114.0242,B 24.9469,C -1.6831,E1 24.9454,E2 199.6964} C_DIS
LIN {X -34.5375,Y -100.3932,Z 104,A -112.473,B 24.9466,C -1.6876,E1 24.9496,E2 198.1315} C_DIS
LIN {X -31.7096,Y -101.3202,Z 104,A -111.0203,B 24.9471,C -1.6803,E1 24.9534,E2 196.6934} C_DIS
LIN {X -29.2135,Y -102.0679,Z 104,A -109.5982,B 24.9471,C -1.68,E1 24.9572,E2 195.2697} C_DIS
LIN {X -25.7876,Y -102.9884,Z 104,A -107.5429,B 24.9468,C -1.6844,E1 24.9628,E2 193.201} C_DIS
LIN {X -23.2615,Y -103.5883,Z 104,A -106.1363,B 24.9468,C -1.6839,E1 24.9666,E2 191.7936} C_DIS
LIN {X -20.7123,Y -104.128,Z 104,A -104.7287,B 24.9468,C -1.6834,E1 24.9705,E2 190.3857} C_DIS
LIN {X -17.7854,Y -104.666,Z 104,A -103.1817,B 24.9471,C -1.6805,E1 24.9747,E2 188.844} C_DIS
LIN {X -14.6548,Y -105.15,Z 104,A -101.5128,B 24.9472,C -1.6785,E1 24.9793,E2 187.1785} C_DIS
LIN {X -11.7021,Y -105.5211,Z 104,A -99.9465,B 24.9473,C -1.6767,E1 24.9837,E2 185.6156} C_DIS
LIN {X -8.7397,Y -105.806,Z 104,A -98.5223,B 24.9478,C -1.6693,E1 24.9876,E2 184.2081} C_DIS
LIN {X -6.1405,Y -105.9886,Z 104,A -97.1166,B 24.9478,C -1.6693,E1 24.9915,E2 182.8019} C_DIS
LIN {X -3.5376,Y -106.1074,Z 104,A -95.7104,B 24.9478,C -1.6694,E1 24.9954,E2 181.3951} C_DIS
LIN {X -1.3028,Y -106.1599,Z 104,A -94.1801,B 24.9469,C -1.6827,E1 24.9998,E2 179.8333} C_DIS
LIN {X -1.3028,Y -106.1599,Z 104,A -94.1801,B 24.9469,C -1.6827,E1 24.9998,E2 179.8333} C_DIS
Enddeposition()
LIN {X 0.729,Y -105.1688,Z 104,A -93.3954,B 24.9466,C -1.6877,E1 25.002,E2 179.0367} C_DIS
Startdeposition()
$VEL.CP = VEL_PRINT
LIN {X -1.8745,Y -105.1604,Z 104,A -95.3928,B 24.9481,C -1.6643,E1 24.9963,E2 181.0895} C_DIS
LIN {X -5.4406,Y -105.0369,Z 104,A -97.3671,B 24.9481,C -1.6629,E1 24.9907,E2 183.0675} C_DIS
LIN {X -8.8811,Y -104.8027,Z 104,A -99.2614,B 24.9482,C -1.6623,E1 24.9855,E2 184.9641} C_DIS
LIN {X -12.3227,Y -104.4527,Z 104,A -101.106,B 24.9482,C -1.6641,E1 24.9804,E2 186.8056} C_DIS
LIN {X -15.912,Y -103.9666,Z 104,A -103.0758,B 24.9481,C -1.6647,E1 24.9749,E2 188.7755} C_DIS
LIN {X -19.196,Y -103.4122,Z 104,A -104.9255,B 24.9481,C -1.6639,E1 24.9698,E2 190.629} C_DIS
LIN {X -22.0034,Y -102.8506,Z 104,A -106.5927,B 24.9483,C -1.6604,E1 24.9652,E2 192.3064} C_DIS
LIN {X -26.1194,Y -101.8823,Z 104,A -108.7899,B 24.948,C -1.6658,E1 24.9593,E2 194.4939} C_DIS
LIN {X -29.1848,Y -101.0482,Z 104,A -110.7043,B 24.9484,C -1.6599,E1 24.9541,E2 196.4255} C_DIS
LIN {X -33.2252,Y -99.7921,Z 104,A -112.8382,B 24.9479,C -1.6682,E1 24.9485,E2 198.5434} C_DIS
LIN {X -36.3705,Y -98.689,Z 104,A -114.568,B 24.9475,C -1.6731,E1 24.9439,E2 200.2651} C_DIS
LIN {X -39.2813,Y -97.5672,Z 104,A -116.5478,B 24.9481,C -1.664,E1 24.9387,E2 202.2706} C_DIS
LIN {X -42.903,Y -96.0295,Z 104,A -118.6303,B 24.9478,C -1.6687,E1 24.9334,E2 204.3471} C_DIS
LIN {X -46.8111,Y -94.1857,Z 104,A -120.8957,B 24.9474,C -1.6749,E1 24.9278,E2 206.6036} C_DIS
LIN {X -50.2957,Y -92.372,Z 104,A -123.0554,B 24.9474,C -1.6769,E1 24.9224,E2 208.7645} C_DIS
LIN {X -53.1438,Y -90.7642,Z 104,A -124.8906,B 24.9473,C -1.6774,E1 24.918,E2 210.6039} C_DIS
LIN {X -56.4468,Y -88.7478,Z 104,A -126.7011,B 24.9464,C -1.6918,E1 24.9137,E2 212.386} C_DIS
LIN {X -58.406,Y -87.4715,Z 104,A -128.0994,B 24.9465,C -1.6891,E1 24.9105,E2 213.7951} C_DIS
LIN {X -61.0497,Y -85.6455,Z 104,A -129.8583,B 24.9464,C -1.6917,E1 24.9064,E2 215.5539} C_DIS
LIN {X -63.6062,Y -83.7661,Z 104,A -131.5839,B 24.9462,C -1.6948,E1 24.9026,E2 217.2782} C_DIS
LIN {X -65.5155,Y -82.2805,Z 104,A -133.079,B 24.9464,C -1.6907,E1 24.8993,E2 218.7887} C_DIS
LIN {X -69.9134,Y -78.5776,Z 104,A -136.0583,B 24.9457,C -1.7023,E1 24.893,E2 221.7518} C_DIS
LIN {X -71.7364,Y -76.9175,Z 104,A -137.5405,B 24.9458,C -1.6999,E1 24.8899,E2 223.2458} C_DIS
LIN {X -73.869,Y -74.8705,Z 104,A -139.4077,B 24.9462,C -1.6939,E1 24.8861,E2 225.1352} C_DIS
LIN {X -76.7729,Y -71.8901,Z 104,A -142.5855,B 24.948,C -1.666,E1 24.88,E2 228.3934} C_DIS
LIN {X -81.0418,Y -67.041,Z 104,A -144.9225,B 24.9448,C -1.7168,E1 24.8759,E2 230.6201} C_DIS
LIN {X -82.7906,Y -64.87,Z 104,A -146.4568,B 24.9446,C -1.7198,E1 24.8733,E2 232.1543} C_DIS
LIN {X -86.1451,Y -60.3439,Z 104,A -149.3152,B 24.9436,C -1.7351,E1 24.8686,E2 234.9903} C_DIS
LIN {X -87.4882,Y -58.3812,Z 104,A -150.9768,B 24.9442,C -1.7251,E1 24.8659,E2 236.684} C_DIS
LIN {X -89.5939,Y -55.095,Z 104,A -153.1063,B 24.9439,C -1.7305,E1 24.8628,E2 238.8113} C_DIS
LIN {X -91.6939,Y -51.5221,Z 104,A -155.4286,B 24.9436,C -1.7343,E1 24.8595,E2 241.1367} C_DIS
LIN {X -93.8243,Y -47.5327,Z 104,A -157.6441,B 24.9426,C -1.75,E1 24.8567,E2 243.3266} C_DIS
LIN {X -95.2546,Y -44.5963,Z 104,A -159.4948,B 24.9424,C -1.7525,E1 24.8545,E2 245.1815} C_DIS
LIN {X -96.6464,Y -41.4974,Z 104,A -161.2697,B 24.9419,C -1.7605,E1 24.8525,E2 246.9471} C_DIS
LIN {X -97.6528,Y -39.0711,Z 104,A -162.9324,B 24.9422,C -1.7563,E1 24.8507,E2 248.629} C_DIS
LIN {X -99.0159,Y -35.4744,Z 104,A -164.9402,B 24.9416,C -1.7656,E1 24.8488,E2 250.6259} C_DIS
LIN {X -99.7718,Y -33.2853,Z 104,A -166.8047,B 24.9427,C -1.748,E1 24.8471,E2 252.543} C_DIS
LIN {X -101.0113,Y -29.3142,Z 104,A -168.5437,B 24.941,C -1.7735,E1 24.8458,E2 254.2312} C_DIS
LIN {X -101.7382,Y -26.6801,Z 104,A -170.5714,B 24.942,C -1.759,E1 24.8443,E2 256.3054} C_DIS
LIN {X -102.6807,Y -22.7823,Z 104,A -172.0338,B 24.9399,C -1.7913,E1 24.8434,E2 257.6992} C_DIS
LIN {X -103.1955,Y -20.3251,Z 104,A -173.6553,B 24.9402,C -1.7866,E1 24.8425,E2 259.3417} C_DIS
LIN {X -103.9125,Y -16.2621,Z 104,A -175.8393,B 24.9395,C -1.7959,E1 24.8415,E2 261.5165} C_DIS
LIN {X -104.4103,Y -12.6853,Z 104,A -177.7298,B 24.9389,C -1.8049,E1 24.8408,E2 263.3969} C_DIS
LIN {X -104.7431,Y -9.5458,Z 104,A -179.4824,B 24.9386,C -1.8092,E1 24.8404,E2 265.1496} C_DIS
LIN {X -104.9988,Y -6.1296,Z 104,A 178.5448,B 24.9385,C -1.8114,E1 24.84,E2 267.1291} C_DIS
LIN {X -105.1368,Y -2.9248,Z 104,A 176.7921,B 24.9381,C -1.8168,E1 24.8398,E2 268.8793} C_DIS
LIN {X -105.1756,Y 0.5899,Z 104,A 175.1172,B 24.9371,C -1.8315,E1 24.8398,E2 270.5293} C_DIS
LIN {X -105.1407,Y 2.7979,Z 104,A 173.6086,B 24.9376,C -1.8246,E1 24.8398,E2 272.0636} C_DIS
LIN {X -104.9597,Y 6.766,Z 104,A 171.4295,B 24.9372,C -1.831,E1 24.8402,E2 274.2404} C_DIS
LIN {X -104.6469,Y 10.5545,Z 104,A 169.3192,B 24.9368,C -1.8363,E1 24.8408,E2 276.3507} C_DIS
LIN {X -104.2481,Y 13.9552,Z 104,A 167.523,B 24.9362,C -1.8448,E1 24.8414,E2 278.1375} C_DIS
LIN {X -103.728,Y 17.3991,Z 104,A 165.6611,B 24.9357,C -1.8521,E1 24.8422,E2 279.9929} C_DIS
LIN {X -103.1371,Y 20.6217,Z 104,A 163.7895,B 24.9355,C -1.8548,E1 24.8432,E2 281.8693} C_DIS
LIN {X -102.5031,Y 23.5658,Z 104,A 162.1842,B 24.9351,C -1.8613,E1 24.8442,E2 283.4685} C_DIS
LIN {X -101.6829,Y 26.8906,Z 104,A 159.999,B 24.9354,C -1.8559,E1 24.8457,E2 285.6793} C_DIS
LIN {X -100.7239,Y 30.2831,Z 104,A 157.1436,B 24.9373,C -1.8294,E1 24.8482,E2 288.6144} C_DIS
LIN {X -98.6294,Y 36.5341,Z 104,A 154.6448,B 24.9338,C -1.8786,E1 24.8504,E2 291.0098} C_DIS
LIN {X -97.2458,Y 40.0708,Z 104,A 152.7622,B 24.9329,C -1.8916,E1 24.8523,E2 292.8721} C_DIS
LIN {X -95.7336,Y 43.5595,Z 104,A 150.5013,B 24.9329,C -1.8911,E1 24.8549,E2 295.1465} C_DIS
LIN {X -94.5873,Y 45.9969,Z 104,A 148.7138,B 24.9334,C -1.8842,E1 24.8571,E2 296.9603} C_DIS
LIN {X -93.1414,Y 48.8563,Z 104,A 147.3144,B 24.9322,C -1.9016,E1 24.8588,E2 298.3256} C_DIS
LIN {X -91.2542,Y 52.2963,Z 104,A 145.2085,B 24.9317,C -1.9089,E1 24.8617,E2 300.425} C_DIS
LIN {X -89.3466,Y 55.4931,Z 104,A 142.7416,B 24.9324,C -1.8992,E1 24.8653,E2 302.9279} C_DIS
LIN {X -87.5048,Y 58.3553,Z 104,A 141.2655,B 24.9311,C -1.9178,E1 24.8676,E2 304.367} C_DIS
LIN {X -85.7658,Y 60.8812,Z 104,A 139.5942,B 24.9307,C -1.9224,E1 24.8702,E2 306.0356} C_DIS
LIN {X -83.4844,Y 63.9739,Z 104,A 137.5905,B 24.9301,C -1.9312,E1 24.8736,E2 308.0278} C_DIS
LIN {X -81.9985,Y 65.8686,Z 104,A 136.0743,B 24.9304,C -1.9274,E1 24.8762,E2 309.5604} C_DIS
LIN {X -79.4262,Y 68.9478,Z 104,A 134.0517,B 24.9295,C -1.9389,E1 24.8799,E2 311.5647} C_DIS
LIN {X -77.4392,Y 71.1715,Z 104,A 132.2965,B 24.9295,C -1.9383,E1 24.8832,E2 313.3292} C_DIS
LIN {X -74.9444,Y 73.7941,Z 104,A 130.3173,B 24.9292,C -1.9429,E1 24.887,E2 315.3059} C_DIS
LIN {X -72.0944,Y 76.5808,Z 104,A 128.2046,B 24.9287,C -1.9501,E1 24.8912,E2 317.41} C_DIS
LIN {X -69.4006,Y 79.0307,Z 104,A 126.1525,B 24.9285,C -1.9522,E1 24.8955,E2 319.4654} C_DIS
LIN {X -66.5079,Y 81.4803,Z 104,A 124.1556,B 24.928,C -1.9593,E1 24.8998,E2 321.4532} C_DIS
LIN {X -63.5053,Y 83.8419,Z 104,A 122.0167,B 24.9279,C -1.9616,E1 24.9045,E2 323.5944} C_DIS
LIN {X -60.6945,Y 85.8989,Z 104,A 120.2239,B 24.9273,C -1.9693,E1 24.9085,E2 325.3751} C_DIS
LIN {X -58.3217,Y 87.5274,Z 104,A 118.45,B 24.9276,C -1.9648,E1 24.9127,E2 327.1655} C_DIS
LIN {X -55.086,Y 89.599,Z 104,A 116.4233,B 24.9271,C -1.9712,E1 24.9175,E2 329.1835} C_DIS
LIN {X -51.9727,Y 91.4401,Z 104,A 114.3699,B 24.9271,C -1.9717,E1 24.9224,E2 331.2418} C_DIS
LIN {X -48.9286,Y 93.1032,Z 104,A 112.6043,B 24.9265,C -1.9795,E1 24.9267,E2 332.9939} C_DIS
LIN {X -45.5096,Y 94.8214,Z 104,A 110.4774,B 24.9265,C -1.9812,E1 24.9321,E2 335.1222} C_DIS
LIN {X -41.6552,Y 96.5776,Z 104,A 108.0934,B 24.9264,C -1.9818,E1 24.9382,E2 337.5105} C_DIS
LIN {X -38.9184,Y 97.713,Z 104,A 106.7248,B 24.9255,C -1.9932,E1 24.9417,E2 338.8551} C_DIS
LIN {X -34.0773,Y 99.5048,Z 104,A 102.6546,B 24.9287,C -1.9503,E1 24.9527,E2 343.0352} C_DIS
LIN {X -28.3847,Y 101.275,Z 104,A 100.4365,B 24.9256,C -1.9919,E1 24.9584,E2 345.1581} C_DIS
LIN {X -25.0703,Y 102.1456,Z 104,A 98.6195,B 24.9253,C -1.9956,E1 24.9633,E2 346.9689} C_DIS
LIN {X -22.3681,Y 102.771,Z 104,A 96.8694,B 24.9259,C -1.988,E1 24.9681,E2 348.7394} C_DIS
LIN {X -17.9628,Y 103.6337,Z 104,A 94.6991,B 24.925,C -2.0002,E1 24.974,E2 350.8829} C_DIS
LIN {X -14.4669,Y 104.1779,Z 104,A 92.6728,B 24.9252,C -1.9978,E1 24.9796,E2 352.9166} C_DIS
LIN {X -11.3494,Y 104.5637,Z 104,A 90.944,B 24.9252,C -1.9981,E1 24.9844,E2 354.6459} C_DIS
LIN {X -8.0193,Y 104.8715,Z 104,A 89.127,B 24.9251,C -1.9991,E1 24.9894,E2 356.4613} C_DIS
LIN {X -4.4459,Y 105.0831,Z 104,A 87.2734,B 24.9247,C -2.0035,E1 24.9946,E2 358.3049} C_DIS
LIN {X -1.0249,Y 105.1728,Z 104,A 85.2917,B 24.925,C -1.9995,E1 25.0001,E2 360.2964} C_DIS
LIN {X 2.8745,Y 105.1384,Z 104,A 83.2156,B 24.9249,C -2.0016,E1 25.0059,E2 362.367} C_DIS
LIN {X 6.4058,Y 104.9835,Z 104,A 81.1881,B 24.9252,C -1.9977,E1 25.0116,E2 364.4031} C_DIS
LIN {X 10.1244,Y 104.6897,Z 104,A 79.1938,B 24.9251,C -1.999,E1 25.0171,E2 366.3932} C_DIS
LIN {X 13.6662,Y 104.2855,Z 104,A 77.3726,B 24.9248,C -2.0033,E1 25.0221,E2 368.2027} C_DIS
LIN {X 16.8791,Y 103.8149,Z 104,A 75.5246,B 24.925,C -1.9997,E1 25.0273,E2 370.0576} C_DIS
LIN {X 20.4423,Y 103.1729,Z 104,A 73.5019,B 24.9252,C -1.9969,E1 25.0328,E2 372.0845} C_DIS
LIN {X 23.123,Y 102.6054,Z 104,A 72.135,B 24.9249,C -2.0011,E1 25.0365,E2 373.4397} C_DIS
LIN {X 26.2518,Y 101.8483,Z 104,A 70.2534,B 24.9254,C -1.995,E1 25.0416,E2 375.3329} C_DIS
LIN {X 30.3178,Y 100.7136,Z 104,A 68.0883,B 24.9251,C -1.9987,E1 25.0474,E2 377.4856} C_DIS
LIN {X 33.6972,Y 99.633,Z 104,A 66.1493,B 24.9252,C -1.9969,E1 25.0526,E2 379.4253} C_DIS
LIN {X 36.3703,Y 98.6891,Z 104,A 64.3246,B 24.9262,C -1.9844,E1 25.0574,E2 381.2757} C_DIS
LIN {X 40.0604,Y 97.2501,Z 104,A 62.5005,B 24.9253,C -1.9954,E1 25.0621,E2 383.0697} C_DIS
LIN {X 43.361,Y 95.8231,Z 104,A 60.406,B 24.9259,C -1.9878,E1 25.0675,E2 385.1771} C_DIS
LIN {X 46.3807,Y 94.3991,Z 104,A 58.6323,B 24.9259,C -1.9874,E1 25.0719,E2 386.9471} C_DIS
LIN {X 49.7531,Y 92.6663,Z 104,A 56.6855,B 24.9258,C -1.9894,E1 25.0767,E2 388.8836} C_DIS
LIN {X 52.8639,Y 90.928,Z 104,A 54.5833,B 24.9265,C -1.9801,E1 25.0818,E2 391.0015} C_DIS
LIN {X 55.6385,Y 89.2557,Z 104,A 53.0711,B 24.9259,C -1.9877,E1 25.0854,E2 392.4911} C_DIS
LIN {X 60.8361,Y 85.7979,Z 104,A 49.7868,B 24.9259,C -1.9868,E1 25.093,E2 395.7665} C_DIS
LIN {X 62.9904,Y 84.2288,Z 104,A 48.0056,B 24.9272,C -1.9709,E1 25.0971,E2 397.579} C_DIS
LIN {X 66.094,Y 81.8158,Z 104,A 45.7828,B 24.9277,C -1.9636,E1 25.1019,E2 399.8107} C_DIS
LIN {X 69.1843,Y 79.2197,Z 104,A 43.8004,B 24.9274,C -1.9681,E1 25.1061,E2 401.7746} C_DIS
LIN {X 72.0158,Y 76.6547,Z 104,A 41.7062,B 24.9277,C -1.9634,E1 25.1104,E2 403.8716} C_DIS
LIN {X 74.3425,Y 74.4028,Z 104,A 39.9037,B 24.9281,C -1.958,E1 25.114,E2 405.6792} C_DIS
LIN {X 76.4765,Y 72.2053,Z 104,A 38.4232,B 24.9278,C -1.9621,E1 25.1169,E2 407.1436} C_DIS
LIN {X 78.9635,Y 69.4776,Z 104,A 36.3829,B 24.9282,C -1.9563,E1 25.1207,E2 409.1885} C_DIS
LIN {X 80.4469,Y 67.7559,Z 104,A 34.9779,B 24.929,C -1.9465,E1 25.1232,E2 410.6102} C_DIS
LIN {X 82.665,Y 65.029,Z 104,A 33.1858,B 24.929,C -1.9471,E1 25.1264,E2 412.3927} C_DIS
LIN {X 84.7839,Y 62.2409,Z 104,A 31.2569,B 24.9293,C -1.9415,E1 25.1296,E2 414.3256} C_DIS
LIN {X 86.709,Y 59.5326,Z 104,A 29.3246,B 24.93,C -1.9318,E1 25.1327,E2 416.2712} C_DIS
LIN {X 89.5451,Y 55.175,Z 104,A 26.1544,B 24.9316,C -1.9104,E1 25.1375,E2 419.4759} C_DIS
LIN {X 91.2932,Y 52.2284,Z 104,A 24.3234,B 24.9318,C -1.9069,E1 25.14,E2 421.3058} C_DIS
LIN {X 92.9501,Y 49.2194,Z 104,A 22.9209,B 24.9308,C -1.9212,E1 25.1418,E2 422.6671} C_DIS
LIN {X 94.4864,Y 46.2046,Z 104,A 21.1545,B 24.9309,C -1.9192,E1 25.144,E2 424.4287} C_DIS
LIN {X 95.9801,Y 43.0125,Z 104,A 18.6897,B 24.933,C -1.891,E1 25.1469,E2 426.9467} C_DIS
LIN {X 97.3785,Y 39.7449,Z 104,A 16.6991,B 24.9335,C -1.8831,E1 25.149,E2 428.9449} C_DIS
LIN {X 98.7628,Y 36.1684,Z 104,A 14.7527,B 24.9335,C -1.8829,E1 25.1509,E2 430.8811} C_DIS
LIN {X 99.8796,Y 32.9634,Z 104,A 13.1964,B 24.9331,C -1.8896,E1 25.1523,E2 432.4128} C_DIS
LIN {X 100.9807,Y 29.4173,Z 104,A 11.2094,B 24.9334,C -1.8849,E1 25.1539,E2 434.3995} C_DIS
LIN {X 102.0123,Y 25.6136,Z 104,A 9.076,B 24.9338,C -1.8789,E1 25.1554,E2 436.5348} C_DIS
LIN {X 102.7643,Y 22.3992,Z 104,A 7.3838,B 24.9338,C -1.8778,E1 25.1564,E2 438.2197} C_DIS
LIN {X 103.4979,Y 18.7191,Z 104,A 5.4503,B 24.934,C -1.8761,E1 25.1574,E2 440.146} C_DIS
LIN {X 104.0331,Y 15.4818,Z 104,A 3.5794,B 24.9347,C -1.8669,E1 25.1582,E2 442.0277} C_DIS
LIN {X 104.4589,Y 12.27,Z 104,A 1.9241,B 24.9347,C -1.8659,E1 25.1588,E2 443.6754} C_DIS
LIN {X 104.7334,Y 9.6504,Z 104,A 0.46,B 24.9351,C -1.8601,E1 25.1592,E2 445.1446} C_DIS
LIN {X 105.0019,Y 6.0734,Z 104,A -1.5381,B 24.9357,C -1.852,E1 25.1596,E2 447.15} C_DIS
LIN {X 105.1497,Y 2.4547,Z 104,A -3.5243,B 24.9362,C -1.845,E1 25.1598,E2 449.1408} C_DIS
LIN {X 105.1722,Y -1.1291,Z 104,A -5.3217,B 24.9362,C -1.8453,E1 25.1598,E2 450.9268} C_DIS
LIN {X 105.0976,Y -4.1085,Z 104,A -8.0231,B 24.9396,C -1.7947,E1 25.1595,E2 453.7315} C_DIS
LIN {X 104.7288,Y -9.7008,Z 104,A -9.9792,B 24.9372,C -1.8309,E1 25.159,E2 455.5905} C_DIS
LIN {X 104.4663,Y -12.2073,Z 104,A -11.9301,B 24.9391,C -1.802,E1 25.1584,E2 457.598} C_DIS
LIN {X 103.976,Y -15.851,Z 104,A -13.9079,B 24.9395,C -1.7966,E1 25.1575,E2 459.5769} C_DIS
LIN {X 103.3627,Y -19.4564,Z 104,A -15.4471,B 24.9386,C -1.8093,E1 25.1568,E2 461.0772} C_DIS
LIN {X 102.7104,Y -22.646,Z 104,A -17.3069,B 24.9393,C -1.8,E1 25.1557,E2 462.9482} C_DIS
LIN {X 101.9542,Y -25.8395,Z 104,A -18.9669,B 24.9393,C -1.7997,E1 25.1546,E2 464.5993} C_DIS
LIN {X 100.9922,Y -29.3786,Z 104,A -21.0346,B 24.9399,C -1.7904,E1 25.153,E2 466.6771} C_DIS
LIN {X 99.8209,Y -33.1398,Z 104,A -23.1618,B 24.9403,C -1.7844,E1 25.1512,E2 468.8063} C_DIS
LIN {X 98.4856,Y -36.9179,Z 104,A -25.1398,B 24.9402,C -1.7863,E1 25.1493,E2 470.7687} C_DIS
LIN {X 96.4799,Y -41.8792,Z 104,A -27.79,B 24.94,C -1.7886,E1 25.1466,E2 473.399} C_DIS
LIN {X 94.4732,Y -46.2311,Z 104,A -31.1663,B 24.9427,C -1.7483,E1 25.1424,E2 476.852} C_DIS
LIN {X 92.9106,Y -49.2945,Z 104,A -32.6081,B 24.9419,C -1.7609,E1 25.1406,E2 478.2566} C_DIS
LIN {X 91.3776,Y -52.0815,Z 104,A -34.0869,B 24.9415,C -1.7666,E1 25.1386,E2 479.7143} C_DIS
LIN {X 89.9348,Y -54.5341,Z 104,A -35.7633,B 24.9422,C -1.7567,E1 25.1362,E2 481.4053} C_DIS
LIN {X 88.2386,Y -57.24,Z 104,A -37.6375,B 24.9429,C -1.7461,E1 25.1334,E2 483.2952} C_DIS
LIN {X 86.3571,Y -60.0388,Z 104,A -39.3038,B 24.9427,C -1.7482,E1 25.1308,E2 484.9483} C_DIS
LIN {X 84.5588,Y -62.5483,Z 104,A -41.0257,B 24.9431,C -1.7418,E1 25.1279,E2 486.6769} C_DIS
LIN {X 81.2643,Y -66.7733,Z 104,A -43.8667,B 24.9434,C -1.7373,E1 25.123,E2 489.5153} C_DIS
LIN {X 76.8598,Y -71.7978,Z 104,A -48.5643,B 24.9469,C -1.6841,E1 25.114,E2 494.3176} C_DIS
LIN {X 72.9405,Y -75.7753,Z 104,A -50.6109,B 24.9447,C -1.7179,E1 25.1101,E2 496.2759} C_DIS
LIN {X 70.9516,Y -77.6411,Z 104,A -52.3805,B 24.9457,C -1.7025,E1 25.1064,E2 498.0745} C_DIS
LIN {X 67.4288,Y -80.7196,Z 104,A -55.1581,B 24.9466,C -1.6873,E1 25.1005,E2 500.8773} C_DIS
LIN {X 64.4579,Y -83.1114,Z 104,A -56.5667,B 24.9452,C -1.7104,E1 25.0975,E2 502.2261} C_DIS
LIN {X 59.6825,Y -86.6047,Z 104,A -60.4932,B 24.9474,C -1.6748,E1 25.0884,E2 506.2231} C_DIS
LIN {X 56.2661,Y -88.8637,Z 104,A -62.2729,B 24.9465,C -1.6889,E1 25.0843,E2 507.9635} C_DIS
LIN {X 52.9982,Y -90.8502,Z 104,A -64.2882,B 24.9466,C -1.6879,E1 25.0795,E2 509.9752} C_DIS
LIN {X 49.9478,Y -92.5607,Z 104,A -66.1033,B 24.9466,C -1.6882,E1 25.0751,E2 511.7841} C_DIS
LIN {X 46.9196,Y -94.1319,Z 104,A -67.9362,B 24.9467,C -1.6862,E1 25.0705,E2 513.6169} C_DIS
LIN {X 44.2696,Y -95.4067,Z 104,A -69.5434,B 24.9469,C -1.6834,E1 25.0664,E2 515.2265} C_DIS
LIN {X 40.9629,Y -96.8725,Z 104,A -71.8675,B 24.948,C -1.6661,E1 25.0604,E2 517.5859} C_DIS
LIN {X 36.3371,Y -98.7012,Z 104,A -73.9568,B 24.9466,C -1.6876,E1 25.0551,E2 519.6199} C_DIS
LIN {X 30.9138,Y -100.5317,Z 104,A -77.3923,B 24.9477,C -1.6708,E1 25.0459,E2 523.0885} C_DIS
LIN {X 28.412,Y -101.2672,Z 104,A -78.907,B 24.948,C -1.6654,E1 25.0418,E2 524.6134} C_DIS
LIN {X 24.5503,Y -102.2724,Z 104,A -81.0004,B 24.948,C -1.6665,E1 25.0361,E2 526.7012} C_DIS
LIN {X 20.9412,Y -103.0715,Z 104,A -82.868,B 24.9477,C -1.6705,E1 25.0311,E2 528.5568} C_DIS
LIN {X 18.3476,Y -103.5648,Z 104,A -84.4588,B 24.9482,C -1.6632,E1 25.0267,E2 530.1631} C_DIS
LIN {X 14.7532,Y -104.1372,Z 104,A -86.3031,B 24.9479,C -1.6674,E1 25.0216,E2 531.9959} C_DIS
LIN {X 11.1619,Y -104.5833,Z 104,A -88.3121,B 24.9481,C -1.6647,E1 25.016,E2 534.0098} C_DIS
LIN {X 7.5234,Y -104.9085,Z 104,A -90.3266,B 24.9481,C -1.6627,E1 25.0104,E2 536.028} C_DIS
LIN {X 4.6508,Y -105.0743,Z 104,A -92.0085,B 24.9485,C -1.6576,E1 25.0057,E2 537.7214} C_DIS
LIN {X 0.729,Y -105.1688,Z 104,A -93.3935,B 24.9467,C -1.6869,E1 25.002,E2 539.0367} C_DIS
Enddeposition()
LIN {X 0.729,Y -105.1688,Z 104,A -93.3935,B 24.9467,C -1.6869,E1 25.002,E2 539.0367} C_DIS
Startdeposition()
$VEL.CP = VEL_PRINT
LIN {X 1.3084,Y -104.1818,Z 104,A -92.7822,B 24.9448,C -1.7156,E1 25.0039,E2 538.3574} C_DIS
LIN {X 4.5231,Y -104.09,Z 104,A -91.1491,B 24.9451,C -1.7109,E1 25.0084,E2 536.736} C_DIS
LIN {X 8.0204,Y -103.8794,Z 104,A -89.1364,B 24.9449,C -1.7152,E1 25.0141,E2 534.7141} C_DIS
LIN {X 11.5495,Y -103.5477,Z 104,A -87.1549,B 24.9447,C -1.7175,E1 25.0196,E2 532.7282} C_DIS
LIN {X 15.1603,Y -103.0806,Z 104,A -85.1834,B 24.9447,C -1.7176,E1 25.025,E2 530.7581} C_DIS
LIN {X 20.2724,Y -102.1986,Z 104,A -82.3493,B 24.9447,C -1.7192,E1 25.0328,E2 527.9235} C_DIS
LIN {X 23.9199,Y -101.4064,Z 104,A -80.2824,B 24.9444,C -1.7217,E1 25.0384,E2 525.8536} C_DIS
LIN {X 29.8017,Y -99.8352,Z 104,A -77.1416,B 24.9448,C -1.7169,E1 25.0469,E2 522.7292} C_DIS
LIN {X 35.0118,Y -98.1305,Z 104,A -73.8274,B 24.9437,C -1.7328,E1 25.0557,E2 519.3837} C_DIS
LIN {X 38.8505,Y -96.6749,Z 104,A -71.4876,B 24.9433,C -1.7393,E1 25.0618,E2 517.0337} C_DIS
LIN {X 42.5873,Y -95.0871,Z 104,A -69.5592,B 24.9439,C -1.7302,E1 25.0667,E2 515.1315} C_DIS
LIN {X 45.4106,Y -93.7719,Z 104,A -67.8615,B 24.9438,C -1.7323,E1 25.071,E2 513.4333} C_DIS
LIN {X 48.5119,Y -92.2051,Z 104,A -65.973,B 24.9436,C -1.7346,E1 25.0757,E2 511.5445} C_DIS
LIN {X 51.404,Y -90.6265,Z 104,A -63.571,B 24.9418,C -1.7623,E1 25.0816,E2 509.0842} C_DIS
LIN {X 54.67,Y -88.6948,Z 104,A -61.9282,B 24.9428,C -1.7477,E1 25.0855,E2 507.481} C_DIS
LIN {X 58.1673,Y -86.4398,Z 104,A -59.4978,B 24.9421,C -1.7582,E1 25.0912,E2 505.0339} C_DIS
LIN {X 62.5985,Y -83.2863,Z 104,A -56.8642,B 24.9426,C -1.7495,E1 25.097,E2 502.43} C_DIS
LIN {X 64.9566,Y -81.4618,Z 104,A -54.4571,B 24.9403,C -1.7853,E1 25.1025,E2 499.9476} C_DIS
LIN {X 68.2978,Y -78.681,Z 104,A -52.0049,B 24.9397,C -1.7934,E1 25.1076,E2 497.4859} C_DIS
LIN {X 71.7841,Y -75.5152,Z 104,A -50.1753,B 24.9415,C -1.7675,E1 25.1112,E2 495.725} C_DIS
LIN {X 76.4807,Y -70.7536,Z 104,A -45.8475,B 24.939,C -1.804,E1 25.1197,E2 491.3295} C_DIS
LIN {X 79.3421,Y -67.5279,Z 104,A -44.19,B 24.9406,C -1.78,E1 25.1226,E2 489.7363} C_DIS
LIN {X 81.8098,Y -64.5164,Z 104,A -41.9835,B 24.9401,C -1.7884,E1 25.1265,E2 487.5202} C_DIS
LIN {X 83.7693,Y -61.9527,Z 104,A -40.2088,B 24.9397,C -1.7932,E1 25.1295,E2 485.7426} C_DIS
LIN {X 85.7215,Y -59.2208,Z 104,A -38.3506,B 24.9393,C -1.7989,E1 25.1325,E2 483.8801} C_DIS
LIN {X 88.0728,Y -55.6657,Z 104,A -36.2439,B 24.9396,C -1.7955,E1 25.1356,E2 481.792} C_DIS
LIN {X 89.4817,Y -53.3703,Z 104,A -34.625,B 24.9389,C -1.8056,E1 25.138,E2 480.1575} C_DIS
LIN {X 91.0592,Y -50.6304,Z 104,A -32.4928,B 24.9374,C -1.8274,E1 25.141,E2 477.9848} C_DIS
LIN {X 92.6297,Y -47.6973,Z 104,A -31.0284,B 24.9381,C -1.8173,E1 25.1428,E2 476.5521} C_DIS
LIN {X 94.6804,Y -43.4853,Z 104,A -28.5628,B 24.9379,C -1.8204,E1 25.1458,E2 474.0926} C_DIS
LIN {X 95.7427,Y -41.0958,Z 104,A -26.7149,B 24.9364,C -1.8422,E1 25.1479,E2 472.2033} C_DIS
LIN {X 97.588,Y -36.496,Z 104,A -24.4759,B 24.9372,C -1.8299,E1 25.1501,E2 470.0057} C_DIS
LIN {X 99.2415,Y -31.7246,Z 104,A -21.792,B 24.9369,C -1.8346,E1 25.1525,E2 467.3258} C_DIS
LIN {X 99.9645,Y -29.3659,Z 104,A -20.3524,B 24.9364,C -1.8424,E1 25.1536,E2 465.8761} C_DIS
LIN {X 100.8672,Y -26.0965,Z 104,A -17.8032,B 24.9339,C -1.8776,E1 25.1555,E2 463.2585} C_DIS
LIN {X 101.8326,Y -22.0305,Z 104,A -16.2821,B 24.9357,C -1.8517,E1 25.1564,E2 461.8073} C_DIS
LIN {X 102.3832,Y -19.3136,Z 104,A -14.4489,B 24.9345,C -1.8698,E1 25.1574,E2 459.9422} C_DIS
LIN {X 103.099,Y -15.0273,Z 104,A -11.9267,B 24.9335,C -1.8832,E1 25.1584,E2 457.4033} C_DIS
LIN {X 103.6267,Y -10.802,Z 104,A -9.934,B 24.934,C -1.8758,E1 25.1591,E2 455.4397} C_DIS
LIN {X 104.0955,Y -4.3941,Z 104,A -6.4597,B 24.9334,C -1.8847,E1 25.1597,E2 451.9651} C_DIS
LIN {X 104.1759,Y -1.6272,Z 104,A -4.8308,B 24.9327,C -1.8942,E1 25.1597,E2 450.3235} C_DIS
LIN {X 104.1654,Y 2.1956,Z 104,A -2.8136,B 24.9325,C -1.8973,E1 25.1597,E2 448.3109} C_DIS
LIN {X 104.0189,Y 5.9412,Z 104,A -0.7289,B 24.932,C -1.905,E1 25.1594,E2 446.2206} C_DIS
LIN {X 103.7523,Y 9.521,Z 104,A 1.1645,B 24.9318,C -1.9079,E1 25.159,E2 444.3316} C_DIS
LIN {X 103.354,Y 13.1599,Z 104,A 3.1795,B 24.9313,C -1.9144,E1 25.1583,E2 442.3131} C_DIS
LIN {X 102.8597,Y 16.5957,Z 104,A 5.1583,B 24.9306,C -1.9233,E1 25.1575,E2 440.3248} C_DIS
LIN {X 102.201,Y 20.2602,Z 104,A 7.1868,B 24.9302,C -1.9289,E1 25.1564,E2 438.295} C_DIS
LIN {X 101.4956,Y 23.5338,Z 104,A 9.3261,B 24.9289,C -1.9474,E1 25.1551,E2 436.1246} C_DIS
LIN {X 100.7057,Y 26.7163,Z 104,A 10.7974,B 24.9295,C -1.9388,E1 25.1541,E2 434.6821} C_DIS
LIN {X 99.6768,Y 30.3318,Z 104,A 13.2938,B 24.9277,C -1.9633,E1 25.152,E2 432.1421} C_DIS
LIN {X 98.5288,Y 33.8769,Z 104,A 15.1349,B 24.9279,C -1.9605,E1 25.1504,E2 430.3179} C_DIS
LIN {X 96.5208,Y 39.2291,Z 104,A 17.9517,B 24.9283,C -1.956,E1 25.1476,E2 427.5275} C_DIS
LIN {X 94.6447,Y 43.5632,Z 104,A 20.6113,B 24.9275,C -1.966,E1 25.1445,E2 424.8587} C_DIS
LIN {X 92.9213,Y 47.1266,Z 104,A 22.9638,B 24.9265,C -1.9795,E1 25.1416,E2 422.4868} C_DIS
LIN {X 89.6886,Y 53.0201,Z 104,A 26.3628,B 24.9267,C -1.977,E1 25.137,E2 419.1113} C_DIS
LIN {X 88.3221,Y 55.2665,Z 104,A 27.7981,B 24.9265,C -1.9804,E1 25.1349,E2 417.6754} C_DIS
LIN {X 86.5619,Y 57.9869,Z 104,A 29.4165,B 24.9266,C -1.9782,E1 25.1324,E2 416.0704} C_DIS
LIN {X 84.8977,Y 60.3952,Z 104,A 31.1615,B 24.9259,C -1.9879,E1 25.1296,E2 414.3109} C_DIS
LIN {X 81.9573,Y 64.3297,Z 104,A 33.6205,B 24.9262,C -1.9844,E1 25.1255,E2 411.8718} C_DIS
LIN {X 79.6576,Y 67.1576,Z 104,A 35.7101,B 24.9255,C -1.9927,E1 25.1217,E2 409.7723} C_DIS
LIN {X 77.7405,Y 69.3659,Z 104,A 38.2079,B 24.9225,C -2.0333,E1 25.1169,E2 407.1897} C_DIS
LIN {X 74.5179,Y 72.8188,Z 104,A 39.9075,B 24.9249,C -2.0017,E1 25.1138,E2 405.5721} C_DIS
LIN {X 72.4708,Y 74.8547,Z 104,A 42.2707,B 24.9222,C -2.0371,E1 25.1089,E2 403.1351} C_DIS
LIN {X 69.3615,Y 77.7444,Z 104,A 43.8689,B 24.9241,C -2.0115,E1 25.1058,E2 401.6039} C_DIS
LIN {X 66.8435,Y 79.9202,Z 104,A 46.2305,B 24.9222,C -2.0368,E1 25.1006,E2 399.1916} C_DIS
LIN {X 64.0662,Y 82.1648,Z 104,A 47.9121,B 24.9228,C -2.0288,E1 25.097,E2 397.5352} C_DIS
LIN {X 60.7546,Y 84.6413,Z 104,A 49.7224,B 24.9239,C -2.0139,E1 25.093,E2 395.7665} C_DIS
LIN {X 58.0256,Y 86.5347,Z 104,A 51.9839,B 24.9224,C -2.0346,E1 25.0877,E2 393.4637} C_DIS
LIN {X 55.5624,Y 88.1373,Z 104,A 53.4794,B 24.9226,C -2.0322,E1 25.0842,E2 391.9787} C_DIS
LIN {X 52.6828,Y 89.888,Z 104,A 55.4,B 24.9221,C -2.0377,E1 25.0795,E2 390.0511} C_DIS
LIN {X 49.6504,Y 91.5971,Z 104,A 57.132,B 24.9225,C -2.033,E1 25.0754,E2 388.3353} C_DIS
LIN {X 46.7958,Y 93.0896,Z 104,A 59.0176,B 24.922,C -2.0398,E1 25.0706,E2 386.4386} C_DIS
LIN {X 43.6997,Y 94.5812,Z 104,A 60.7587,B 24.9223,C -2.0362,E1 25.0663,E2 384.7108} C_DIS
LIN {X 39.8351,Y 96.2741,Z 104,A 63.028,B 24.9223,C -2.0366,E1 25.0605,E2 382.4458} C_DIS
LIN {X 34.9348,Y 98.1578,Z 104,A 66.3029,B 24.9208,C -2.0548,E1 25.0518,E2 379.1347} C_DIS
LIN {X 30.9644,Y 99.4807,Z 104,A 68.3518,B 24.9215,C -2.0466,E1 25.0464,E2 377.109} C_DIS
LIN {X 25.445,Y 101.0346,Z 104,A 71.3764,B 24.9217,C -2.0436,E1 25.0383,E2 374.0965} C_DIS
LIN {X 21.6572,Y 101.9139,Z 104,A 73.7026,B 24.921,C -2.0521,E1 25.0319,E2 371.7533} C_DIS
LIN {X 18.0876,Y 102.6068,Z 104,A 75.6374,B 24.9212,C -2.0503,E1 25.0266,E2 369.8249} C_DIS
LIN {X 14.6719,Y 103.15,Z 104,A 77.4809,B 24.9213,C -2.0486,E1 25.0215,E2 367.9872} C_DIS
LIN {X 11.0703,Y 103.5987,Z 104,A 79.4945,B 24.9213,C -2.0496,E1 25.016,E2 365.9726} C_DIS
LIN {X 7.6736,Y 103.9072,Z 104,A 81.4775,B 24.9209,C -2.0539,E1 25.0104,E2 363.9805} C_DIS
LIN {X 4.2439,Y 104.102,Z 104,A 83.2825,B 24.9211,C -2.0506,E1 25.0054,E2 362.1839} C_DIS
LIN {X 0.6909,Y 104.1859,Z 104,A 85.1859,B 24.9213,C -2.0483,E1 25.0001,E2 360.2862} C_DIS
LIN {X -2.3121,Y 104.1633,Z 104,A 86.936,B 24.9211,C -2.0517,E1 24.9952,E2 358.528} C_DIS
LIN {X -6.0433,Y 104.0132,Z 104,A 89.0313,B 24.921,C -2.0526,E1 24.9893,E2 356.43} C_DIS
LIN {X -9.7522,Y 103.7309,Z 104,A 91.0632,B 24.9211,C -2.0511,E1 24.9837,E2 354.4007} C_DIS
LIN {X -13.5447,Y 103.3042,Z 104,A 93.016,B 24.9216,C -2.0443,E1 24.9783,E2 352.4626} C_DIS
LIN {X -16.1013,Y 102.9367,Z 104,A 94.5569,B 24.9214,C -2.0479,E1 24.974,E2 350.9118} C_DIS
LIN {X -20.6302,Y 102.1258,Z 104,A 97.2473,B 24.921,C -2.052,E1 24.9666,E2 348.2089} C_DIS
LIN {X -26.1698,Y 100.8483,Z 104,A 100.0837,B 24.9221,C -2.0381,E1 24.959,E2 345.4016} C_DIS
LIN {X -29.4221,Y 99.9476,Z 104,A 102.6174,B 24.9203,C -2.0617,E1 24.9521,E2 342.8077} C_DIS
LIN {X -33.2289,Y 98.7473,Z 104,A 104.0718,B 24.9226,C -2.0312,E1 24.9484,E2 341.4232} C_DIS
LIN {X -35.5898,Y 97.9212,Z 104,A 105.6554,B 24.9222,C -2.0372,E1 24.9442,E2 339.8222} C_DIS
LIN {X -39.4504,Y 96.4307,Z 104,A 107.8676,B 24.9226,C -2.0317,E1 24.9384,E2 337.6182} C_DIS
LIN {X -41.8231,Y 95.4257,Z 104,A 109.7578,B 24.9214,C -2.0473,E1 24.9335,E2 335.6865} C_DIS
LIN {X -44.9318,Y 94.0019,Z 104,A 111.169,B 24.923,C -2.0269,E1 24.9301,E2 334.3202} C_DIS
LIN {X -47.3595,Y 92.8023,Z 104,A 112.7022,B 24.923,C -2.0261,E1 24.9262,E2 332.7848} C_DIS
LIN {X -50.4671,Y 91.1504,Z 104,A 115.0929,B 24.922,C -2.0396,E1 24.9203,E2 330.355} C_DIS
LIN {X -53.5157,Y 89.3957,Z 104,A 116.6653,B 24.9233,C -2.0227,E1 24.9166,E2 328.8181} C_DIS
LIN {X -56.8228,Y 87.3309,Z 104,A 118.7757,B 24.9237,C -2.0174,E1 24.9116,E2 326.7136} C_DIS
LIN {X -59.7622,Y 85.3451,Z 104,A 120.6665,B 24.9241,C -2.0113,E1 24.9073,E2 324.8309} C_DIS
LIN {X -62.4601,Y 83.3903,Z 104,A 123.0384,B 24.9229,C -2.0273,E1 24.9019,E2 322.4124} C_DIS
LIN {X -65.3659,Y 81.1331,Z 104,A 124.3695,B 24.9252,C -1.9976,E1 24.8991,E2 321.1472} C_DIS
LIN {X -67.4928,Y 79.372,Z 104,A 126.0814,B 24.9249,C -2.0012,E1 24.8954,E2 319.42} C_DIS
LIN {X -70.0782,Y 77.1004,Z 104,A 128.0656,B 24.9249,C -2.0002,E1 24.8913,E2 317.4303} C_DIS
LIN {X -72.5135,Y 74.8135,Z 104,A 129.9286,B 24.9252,C -1.9968,E1 24.8875,E2 315.5678} C_DIS
LIN {X -75.1713,Y 72.1423,Z 104,A 131.9576,B 24.9257,C -1.9902,E1 24.8836,E2 313.5459} C_DIS
LIN {X -77.7012,Y 69.4098,Z 104,A 133.922,B 24.9263,C -1.982,E1 24.8799,E2 311.5923} C_DIS
LIN {X -79.9901,Y 66.7594,Z 104,A 136.4311,B 24.9251,C -1.9981,E1 24.8753,E2 309.0332} C_DIS
LIN {X -82.3105,Y 63.8772,Z 104,A 138.0162,B 24.9268,C -1.9764,E1 24.8727,E2 307.4923} C_DIS
LIN {X -84.5048,Y 60.9459,Z 104,A 140.0509,B 24.9271,C -1.9717,E1 24.8693,E2 305.4591} C_DIS
LIN {X -87.2542,Y 56.9396,Z 104,A 142.8447,B 24.9273,C -1.9686,E1 24.8649,E2 302.6587} C_DIS
LIN {X -90.8648,Y 50.9786,Z 104,A 146.2229,B 24.9293,C -1.9413,E1 24.8602,E2 299.3281} C_DIS
LIN {X -93.7641,Y 45.4267,Z 104,A 149.7552,B 24.9299,C -1.9341,E1 24.8557,E2 295.794} C_DIS
LIN {X -95.6811,Y 41.2371,Z 104,A 152.4759,B 24.9299,C -1.9331,E1 24.8525,E2 293.0609} C_DIS
LIN {X -96.9163,Y 38.2419,Z 104,A 154.3274,B 24.9302,C -1.9301,E1 24.8506,E2 291.2062} C_DIS
LIN {X -98.7215,Y 33.3052,Z 104,A 157.2887,B 24.9306,C -1.9237,E1 24.8478,E2 288.2435} C_DIS
LIN {X -99.6886,Y 30.2939,Z 104,A 159.1212,B 24.9308,C -1.9215,E1 24.8463,E2 286.4056} C_DIS
LIN {X -100.767,Y 26.4847,Z 104,A 161.052,B 24.9319,C -1.9059,E1 24.8449,E2 284.5009} C_DIS
LIN {X -101.3445,Y 24.1816,Z 104,A 162.3836,B 24.9321,C -1.9026,E1 24.844,E2 283.1692} C_DIS
LIN {X -102.2188,Y 20.1673,Z 104,A 164.8554,B 24.9321,C -1.9029,E1 24.8425,E2 280.6821} C_DIS
LIN {X -102.8366,Y 16.7342,Z 104,A 167.1147,B 24.9317,C -1.9089,E1 24.8415,E2 278.3951} C_DIS
LIN {X -103.472,Y 12.1957,Z 104,A 169.5547,B 24.9325,C -1.898,E1 24.8407,E2 275.9667} C_DIS
LIN {X -103.8122,Y 8.861,Z 104,A 171.1725,B 24.9335,C -1.8839,E1 24.8403,E2 274.3728} C_DIS
LIN {X -104.0315,Y 5.7131,Z 104,A 172.8923,B 24.9339,C -1.8778,E1 24.84,E2 272.6572} C_DIS
LIN {X -104.1801,Y 1.4007,Z 104,A 175.3479,B 24.9342,C -1.873,E1 24.8398,E2 270.1981} C_DIS
LIN {X -104.161,Y -2.435,Z 104,A 177.3035,B 24.9351,C -1.8608,E1 24.8398,E2 268.26} C_DIS
LIN {X -104.0425,Y -5.5139,Z 104,A 179.1382,B 24.9351,C -1.8603,E1 24.8401,E2 266.4153} C_DIS
LIN {X -103.7437,Y -9.6139,Z 104,A -178.5539,B 24.9355,C -1.8548,E1 24.8406,E2 264.1067} C_DIS
LIN {X -103.215,Y -14.2145,Z 104,A -176.0012,B 24.9361,C -1.8469,E1 24.8415,E2 261.5577} C_DIS
LIN {X -102.6532,Y -17.8292,Z 104,A -173.653,B 24.9357,C -1.8526,E1 24.8426,E2 259.1818} C_DIS
LIN {X -101.7731,Y -22.3031,Z 104,A -170.9605,B 24.9357,C -1.8515,E1 24.8442,E2 256.4761} C_DIS
LIN {X -100.875,Y -26.0659,Z 104,A -169.4223,B 24.9377,C -1.8238,E1 24.8452,E2 254.9951} C_DIS
LIN {X -99.8671,Y -29.6943,Z 104,A -166.869,B 24.9369,C -1.8348,E1 24.8472,E2 252.4006} C_DIS
LIN {X -98.8526,Y -32.9167,Z 104,A -165.6448,B 24.9388,C -1.8064,E1 24.8482,E2 251.2372} C_DIS
LIN {X -97.9002,Y -35.6475,Z 104,A -163.8616,B 24.9387,C -1.8086,E1 24.8499,E2 249.4385} C_DIS
LIN {X -96.7279,Y -38.7202,Z 104,A -161.5321,B 24.9378,C -1.8222,E1 24.8524,E2 247.0638} C_DIS
LIN {X -95.3998,Y -41.8824,Z 104,A -160.0311,B 24.9391,C -1.8028,E1 24.854,E2 245.6007} C_DIS
LIN {X -93.8752,Y -45.1955,Z 104,A -158.0609,B 24.9396,C -1.7959,E1 24.8563,E2 243.6363} C_DIS
LIN {X -90.9745,Y -50.782,Z 104,A -154.658,B 24.9403,C -1.7842,E1 24.8608,E2 240.2432} C_DIS
LIN {X -89.375,Y -53.5505,Z 104,A -152.6276,B 24.94,C -1.7894,E1 24.8637,E2 238.19} C_DIS
LIN {X -87.3622,Y -56.7749,Z 104,A -150.7234,B 24.9408,C -1.7771,E1 24.8665,E2 236.3052} C_DIS
LIN {X -85.6646,Y -59.3026,Z 104,A -148.723,B 24.9403,C -1.7849,E1 24.8697,E2 234.2765} C_DIS
LIN {X -82.7964,Y -63.2466,Z 104,A -146.5494,B 24.942,C -1.7596,E1 24.8733,E2 232.1525} C_DIS
LIN {X -81.2817,Y -65.1825,Z 104,A -144.9332,B 24.9415,C -1.7661,E1 24.8761,E2 230.5134} C_DIS
LIN {X -77.1986,Y -69.9688,Z 104,A -141.4331,B 24.942,C -1.7596,E1 24.8825,E2 227.0128} C_DIS
LIN {X -75.0113,Y -72.3083,Z 104,A -139.7646,B 24.9424,C -1.7524,E1 24.8857,E2 225.3545} C_DIS
LIN {X -72.6639,Y -74.6686,Z 104,A -138.0379,B 24.943,C -1.7446,E1 24.8891,E2 223.6389} C_DIS
LIN {X -70.4635,Y -76.7469,Z 104,A -136.2608,B 24.943,C -1.7454,E1 24.8928,E2 221.8525} C_DIS
LIN {X -67.5875,Y -79.2913,Z 104,A -134.0991,B 24.943,C -1.7432,E1 24.8973,E2 219.6878} C_DIS
LIN {X -64.398,Y -81.9033,Z 104,A -131.8929,B 24.9435,C -1.7367,E1 24.9021,E2 217.4888} C_DIS
LIN {X -61.8123,Y -83.8721,Z 104,A -130.0337,B 24.9435,C -1.7362,E1 24.9063,E2 215.624} C_DIS
LIN {X -58.9237,Y -85.9273,Z 104,A -127.6576,B 24.9427,C -1.7491,E1 24.9118,E2 213.2093} C_DIS
LIN {X -56.2037,Y -87.7288,Z 104,A -126.2632,B 24.9438,C -1.7312,E1 24.915,E2 211.8529} C_DIS
LIN {X -52.2408,Y -90.1456,Z 104,A -123.6897,B 24.944,C -1.7282,E1 24.9212,E2 209.2785} C_DIS
LIN {X -49.0757,Y -91.9082,Z 104,A -121.6435,B 24.944,C -1.7276,E1 24.9262,E2 207.2281} C_DIS
LIN {X -45.8363,Y -93.5652,Z 104,A -119.3508,B 24.9435,C -1.7363,E1 24.932,E2 204.9087} C_DIS
LIN {X -41.6631,Y -95.4954,Z 104,A -117.2069,B 24.9446,C -1.7188,E1 24.9374,E2 202.8013} C_DIS
LIN {X -37.8063,Y -97.0874,Z 104,A -114.6684,B 24.9442,C -1.7258,E1 24.944,E2 200.2403} C_DIS
LIN {X -33.663,Y -98.6009,Z 104,A -112.4291,B 24.9448,C -1.7166,E1 24.9499,E2 198.0187} C_DIS
LIN {X -28.4413,Y -100.2311,Z 104,A -109.554,B 24.9452,C -1.7092,E1 24.9575,E2 195.156} C_DIS
LIN {X -25.1785,Y -101.1013,Z 104,A -107.523,B 24.9449,C -1.7149,E1 24.963,E2 193.1087} C_DIS
LIN {X -21.9617,Y -101.8476,Z 104,A -105.7373,B 24.945,C -1.7128,E1 24.9679,E2 191.3255} C_DIS
LIN {X -18.4097,Y -102.5488,Z 104,A -103.7712,B 24.9451,C -1.7111,E1 24.9733,E2 189.3614} C_DIS
LIN {X -14.7667,Y -103.1365,Z 104,A -101.7486,B 24.9451,C -1.7103,E1 24.9789,E2 187.3389} C_DIS
LIN {X -11.077,Y -103.598,Z 104,A -99.6914,B 24.9451,C -1.7105,E1 24.9846,E2 185.28} C_DIS
LIN {X -7.8744,Y -103.8911,Z 104,A -97.8652,B 24.9451,C -1.7127,E1 24.9897,E2 183.4477} C_DIS
LIN {X -4.3414,Y -104.0978,Z 104,A -95.9575,B 24.9451,C -1.7114,E1 24.995,E2 181.5427} C_DIS
LIN {X -0.5577,Y -104.1868,Z 104,A -93.8983,B 24.9451,C -1.7109,E1 25.0007,E2 179.4847} C_DIS
LIN {X -0.5577,Y -104.1868,Z 104,A -93.8983,B 24.9451,C -1.7109,E1 25.0007,E2 179.4847} C_DIS
Enddeposition()
LIN {X 0.7163,Y -103.1921,Z 104,A -93.48,B 24.9447,C -1.7172,E1 25.002,E2 179.0514} C_DIS
Startdeposition()
$VEL.CP = VEL_PRINT
LIN {X -1.9414,Y -103.1811,Z 104,A -95.5481,B 24.9462,C -1.6938,E1 24.996,E2 181.175} C_DIS
LIN {X -5.6012,Y -103.0473,Z 104,A -97.596,B 24.9462,C -1.6931,E1 24.9903,E2 183.2251} C_DIS
LIN {X -9.172,Y -102.7914,Z 104,A -99.5703,B 24.9462,C -1.6936,E1 24.9848,E2 185.199} C_DIS
LIN {X -12.5555,Y -102.4342,Z 104,A -101.4102,B 24.9462,C -1.6957,E1 24.9797,E2 187.035} C_DIS
LIN {X -15.65,Y -102.0059,Z 104,A -103.2133,B 24.9462,C -1.6935,E1 24.9747,E2 188.8448} C_DIS
LIN {X -18.9351,Y -101.4491,Z 104,A -105.1743,B 24.9465,C -1.6899,E1 24.9693,E2 190.8164} C_DIS
LIN {X -22.7608,Y -100.6592,Z 104,A -107.2083,B 24.9461,C -1.696,E1 24.9638,E2 192.8383} C_DIS
LIN {X -26.9137,Y -99.6281,Z 104,A -109.3155,B 24.9454,C -1.7075,E1 24.9581,E2 194.9212} C_DIS
LIN {X -31.9131,Y -98.1411,Z 104,A -112.2272,B 24.9453,C -1.7089,E1 24.9504,E2 197.8345} C_DIS
LIN {X -36.6802,Y -96.4608,Z 104,A -115.3962,B 24.946,C -1.6978,E1 24.942,E2 201.0363} C_DIS
LIN {X -40.242,Y -95.0301,Z 104,A -117.4051,B 24.9456,C -1.7045,E1 24.9368,E2 203.0338} C_DIS
LIN {X -42.7259,Y -93.94,Z 104,A -119.6493,B 24.9472,C -1.679,E1 24.9309,E2 205.3441} C_DIS
LIN {X -46.6721,Y -92.0431,Z 104,A -121.3624,B 24.9453,C -1.7083,E1 24.9268,E2 206.992} C_DIS
LIN {X -49.5185,Y -90.5436,Z 104,A -122.9929,B 24.9448,C -1.7164,E1 24.9228,E2 208.6078} C_DIS
LIN {X -53.0623,Y -88.5149,Z 104,A -125.5439,B 24.9453,C -1.7092,E1 24.9166,E2 211.1837} C_DIS
LIN {X -55.7616,Y -86.8375,Z 104,A -127.9195,B 24.9465,C -1.6898,E1 24.9109,E2 213.6132} C_DIS
LIN {X -59.4501,Y -84.3572,Z 104,A -129.7793,B 24.9448,C -1.7158,E1 24.9068,E2 215.4173} C_DIS
LIN {X -61.9245,Y -82.5559,Z 104,A -131.4014,B 24.9445,C -1.7216,E1 24.9031,E2 217.0314} C_DIS
LIN {X -64.9242,Y -80.2182,Z 104,A -133.529,B 24.9442,C -1.7249,E1 24.8985,E2 219.1591} C_DIS
LIN {X -68.3843,Y -77.292,Z 104,A -136.1712,B 24.9442,C -1.7251,E1 24.8929,E2 221.8109} C_DIS
LIN {X -70.9959,Y -74.8989,Z 104,A -137.8289,B 24.9432,C -1.7403,E1 24.8895,E2 223.4393} C_DIS
LIN {X -73.0999,Y -72.8472,Z 104,A -139.7167,B 24.9436,C -1.7345,E1 24.8857,E2 225.3489} C_DIS
LIN {X -75.5767,Y -70.2753,Z 104,A -141.5389,B 24.943,C -1.7446,E1 24.8823,E2 227.155} C_DIS
LIN {X -79.2647,Y -66.085,Z 104,A -144.7697,B 24.9428,C -1.747,E1 24.8763,E2 230.3947} C_DIS
LIN {X -80.9801,Y -63.9713,Z 104,A -146.1965,B 24.9424,C -1.7536,E1 24.8738,E2 231.8125} C_DIS
LIN {X -83.8167,Y -60.2077,Z 104,A -149.0607,B 24.9425,C -1.7512,E1 24.8691,E2 234.6962} C_DIS
LIN {X -86.0819,Y -56.9213,Z 104,A -151.0739,B 24.9417,C -1.764,E1 24.8659,E2 236.6887} C_DIS
LIN {X -87.974,Y -53.9524,Z 104,A -153.1845,B 24.9417,C -1.7636,E1 24.8628,E2 238.8111} C_DIS
LIN {X -89.8508,Y -50.7662,Z 104,A -155.0272,B 24.9408,C -1.7765,E1 24.8602,E2 240.6326} C_DIS
LIN {X -93.247,Y -44.2196,Z 104,A -159.2017,B 24.9403,C -1.785,E1 24.8549,E2 244.8092} C_DIS
LIN {X -95.8037,Y -38.368,Z 104,A -162.9581,B 24.9401,C -1.7878,E1 24.8508,E2 248.5797} C_DIS
LIN {X -97.0937,Y -34.9728,Z 104,A -164.9501,B 24.9396,C -1.7946,E1 24.8488,E2 250.5668} C_DIS
LIN {X -97.9391,Y -32.5309,Z 104,A -166.8823,B 24.9405,C -1.7816,E1 24.8471,E2 252.541} C_DIS
LIN {X -99.0475,Y -28.9801,Z 104,A -168.5172,B 24.9391,C -1.8028,E1 24.8458,E2 254.1349} C_DIS
LIN {X -99.745,Y -26.4808,Z 104,A -170.3815,B 24.9398,C -1.7925,E1 24.8445,E2 256.0345} C_DIS
LIN {X -100.6025,Y -23.0062,Z 104,A -171.8267,B 24.9381,C -1.8174,E1 24.8436,E2 257.4288} C_DIS
LIN {X -101.786,Y -17.0211,Z 104,A -175.2631,B 24.9375,C -1.8263,E1 24.8418,E2 260.8643} C_DIS
LIN {X -102.2778,Y -13.7699,Z 104,A -176.9655,B 24.9368,C -1.8363,E1 24.8411,E2 262.5531} C_DIS
LIN {X -102.7444,Y -9.682,Z 104,A -179.8274,B 24.9377,C -1.8236,E1 24.8403,E2 265.4623} C_DIS
LIN {X -103.0028,Y -6.3915,Z 104,A 178.7051,B 24.9364,C -1.842,E1 24.84,E2 266.8947} C_DIS
LIN {X -103.1557,Y -3.0044,Z 104,A 176.9096,B 24.9358,C -1.8511,E1 24.8398,E2 268.6793} C_DIS
LIN {X -103.1935,Y 1.2645,Z 104,A 173.8932,B 24.9368,C -1.8365,E1 24.8398,E2 271.7487} C_DIS
LIN {X -103.0771,Y 5.0573,Z 104,A 172.234,B 24.9352,C -1.8587,E1 24.8401,E2 273.3651} C_DIS
LIN {X -102.8712,Y 8.2233,Z 104,A 169.904,B 24.9362,C -1.8449,E1 24.8406,E2 275.742} C_DIS
LIN {X -102.4514,Y 12.4087,Z 104,A 168.346,B 24.9338,C -1.8791,E1 24.8411,E2 277.2277} C_DIS
LIN {X -101.6544,Y 17.7968,Z 104,A 165.0938,B 24.9337,C -1.8809,E1 24.8425,E2 280.4949} C_DIS
LIN {X -101.0089,Y 21.1534,Z 104,A 163.394,B 24.9328,C -1.8938,E1 24.8434,E2 282.1739} C_DIS
LIN {X -100.5099,Y 23.4073,Z 104,A 162.1959,B 24.9323,C -1.9008,E1 24.8441,E2 283.3624} C_DIS
LIN {X -99.714,Y 26.5959,Z 104,A 160.0791,B 24.9326,C -1.8965,E1 24.8456,E2 285.5019} C_DIS
LIN {X -98.7457,Y 29.9958,Z 104,A 158.0642,B 24.9323,C -1.9008,E1 24.8472,E2 287.5181} C_DIS
LIN {X -97.8184,Y 32.8888,Z 104,A 155.7559,B 24.9334,C -1.8848,E1 24.8493,E2 289.8777} C_DIS
LIN {X -96.3428,Y 36.9918,Z 104,A 153.995,B 24.9313,C -1.9149,E1 24.8509,E2 291.5768} C_DIS
LIN {X -94.9888,Y 40.34,Z 104,A 151.3968,B 24.9323,C -1.9006,E1 24.8538,E2 294.2234} C_DIS
LIN {X -93.3699,Y 43.9587,Z 104,A 149.8912,B 24.9301,C -1.9312,E1 24.8555,E2 295.6643} C_DIS
LIN {X -91.4976,Y 47.7331,Z 104,A 147.2388,B 24.9304,C -1.9273,E1 24.8589,E2 298.3403} C_DIS
LIN {X -89.6574,Y 51.1057,Z 104,A 144.989,B 24.9302,C -1.9295,E1 24.8619,E2 300.5967} C_DIS
LIN {X -87.3967,Y 54.8815,Z 104,A 143.0477,B 24.9284,C -1.9539,E1 24.8647,E2 302.4897} C_DIS
LIN {X -84.4069,Y 59.3795,Z 104,A 139.7039,B 24.9287,C -1.9502,E1 24.87,E2 305.859} C_DIS
LIN {X -82.3427,Y 62.2082,Z 104,A 136.9501,B 24.9304,C -1.9274,E1 24.8747,E2 308.6803} C_DIS
LIN {X -79.1684,Y 66.201,Z 104,A 134.9294,B 24.9278,C -1.9629,E1 24.8782,E2 310.6257} C_DIS
LIN {X -76.9073,Y 68.8141,Z 104,A 133.045,B 24.9273,C -1.969,E1 24.8816,E2 312.5041} C_DIS
LIN {X -74.5388,Y 71.3736,Z 104,A 131.1136,B 24.9269,C -1.974,E1 24.8853,E2 314.4321} C_DIS
LIN {X -72.1596,Y 73.7791,Z 104,A 129.1415,B 24.9269,C -1.9752,E1 24.8892,E2 316.4095} C_DIS
LIN {X -69.8575,Y 75.9609,Z 104,A 127.5075,B 24.9262,C -1.9838,E1 24.8925,E2 318.0297} C_DIS
LIN {X -67.3573,Y 78.1884,Z 104,A 125.5404,B 24.9262,C -1.9842,E1 24.8967,E2 320.0036} C_DIS
LIN {X -65.3901,Y 79.8406,Z 104,A 123.1396,B 24.9285,C -1.9531,E1 24.9021,E2 322.4874} C_DIS
LIN {X -61.0092,Y 83.2345,Z 104,A 121.0538,B 24.9254,C -1.9944,E1 24.9065,E2 324.4824} C_DIS
LIN {X -57.9121,Y 85.4184,Z 104,A 118.9505,B 24.9251,C -1.9986,E1 24.9113,E2 326.5828} C_DIS
LIN {X -55.7382,Y 86.8525,Z 104,A 117.2113,B 24.9257,C -1.991,E1 24.9155,E2 328.3459} C_DIS
LIN {X -48.903,Y 90.8775,Z 104,A 112.1451,B 24.9268,C -1.9752,E1 24.9279,E2 333.4644} C_DIS
LIN {X -44.1634,Y 93.274,Z 104,A 109.8002,B 24.9249,C -2.0013,E1 24.9337,E2 335.7531} C_DIS
LIN {X -39.6095,Y 95.2967,Z 104,A 107.2586,B 24.924,C -2.0135,E1 24.9401,E2 338.2719} C_DIS
LIN {X -37.132,Y 96.2897,Z 104,A 105.574,B 24.9244,C -2.0081,E1 24.9446,E2 339.9728} C_DIS
LIN {X -32.3666,Y 97.9942,Z 104,A 102.4448,B 24.925,C -2,E1 24.9529,E2 343.1271} C_DIS
LIN {X -28.6201,Y 99.1527,Z 104,A 100.8106,B 24.9233,C -2.0222,E1 24.9572,E2 344.7115} C_DIS
LIN {X -25.7593,Y 99.9328,Z 104,A 98.8482,B 24.9241,C -2.0123,E1 24.9625,E2 346.7003} C_DIS
LIN {X -21.4215,Y 100.9533,Z 104,A 96.1869,B 24.9244,C -2.0076,E1 24.9698,E2 349.3761} C_DIS
LIN {X -17.7731,Y 101.6586,Z 104,A 94.565,B 24.9231,C -2.0253,E1 24.9742,E2 350.9574} C_DIS
LIN {X -14.4804,Y 102.1784,Z 104,A 92.8839,B 24.9225,C -2.0329,E1 24.9788,E2 352.622} C_DIS
LIN {X -10.3809,Y 102.6766,Z 104,A 90.4972,B 24.9227,C -2.0307,E1 24.9854,E2 355.0155} C_DIS
LIN {X -6.8405,Y 102.9725,Z 104,A 88.5744,B 24.9225,C -2.0334,E1 24.9907,E2 356.9327} C_DIS
LIN {X -3.4739,Y 103.1413,Z 104,A 86.5801,B 24.9228,C -2.0294,E1 24.9963,E2 358.9368} C_DIS
LIN {X 0.2036,Y 103.2,Z 104,A 84.5593,B 24.9227,C -2.0306,E1 25.002,E2 360.9546} C_DIS
LIN {X 3.7986,Y 103.1314,Z 104,A 82.5046,B 24.9228,C -2.0286,E1 25.0077,E2 363.0137} C_DIS
LIN {X 7.1375,Y 102.9524,Z 104,A 80.8006,B 24.9224,C -2.0344,E1 25.0124,E2 364.7033} C_DIS
LIN {X 10.6471,Y 102.6487,Z 104,A 78.8215,B 24.9224,C -2.0333,E1 25.0179,E2 366.6838} C_DIS
LIN {X 14.0725,Y 102.2363,Z 104,A 76.8076,B 24.9228,C -2.0292,E1 25.0235,E2 368.706} C_DIS
LIN {X 17.5969,Y 101.6897,Z 104,A 74.8882,B 24.9227,C -2.0308,E1 25.0288,E2 370.6195} C_DIS
LIN {X 21.0024,Y 101.0399,Z 104,A 72.6987,B 24.9235,C -2.0199,E1 25.0349,E2 372.8322} C_DIS
LIN {X 24.6336,Y 100.2164,Z 104,A 70.3445,B 24.9244,C -2.0078,E1 25.0413,E2 375.2118} C_DIS
Enddeposition()
END
